    movel(p[x_c + -0.037960, y_c + 0.070717, z_c, rx, ry, rz], a, v)
    movel(p[x_c + -0.038280, y_c + 0.070511, z_c, rx, ry, rz], a, v)
    movel(p[x_c + -0.038598, y_c + 0.070300, z_c, rx, ry, rz], a, v)
    movel(p[x_c + -0.038913, y_c + 0.070083, z_c, rx, ry, rz], a, v)
    movel(p[x_c + -0.039226, y_c + 0.069859, z_c, rx, ry, rz], a, v)
    movel(p[x_c + -0.039535, y_c + 0.069631, z_c, rx, ry, rz], a, v)
    movel(p[x_c + -0.039842, y_c + 0.069396, z_c, rx, ry, rz], a, v)
    movel(p[x_c + -0.040146, y_c + 0.069155, z_c, rx, ry, rz], a, v)
    movel(p[x_c + -0.040448, y_c + 0.068909, z_c, rx, ry, rz], a, v)
    movel(p[x_c + -0.040746, y_c + 0.068657, z_c, rx, ry, rz], a, v)
    movel(p[x_c + -0.041042, y_c + 0.068400, z_c, rx, ry, rz], a, v)
    movel(p[x_c + -0.041335, y_c + 0.068137, z_c, rx, ry, rz], a, v)
    movel(p[x_c + -0.041625, y_c + 0.067868, z_c, rx, ry, rz], a, v)
    movel(p[x_c + -0.041912, y_c + 0.067594, z_c, rx, ry, rz], a, v)
    movel(p[x_c + -0.042196, y_c + 0.067314, z_c, rx, ry, rz], a, v)
    movel(p[x_c + -0.042477, y_c + 0.067029, z_c, rx, ry, rz], a, v)
    movel(p[x_c + -0.042756, y_c + 0.066738, z_c, rx, ry, rz], a, v)
    movel(p[x_c + -0.043031, y_c + 0.066441, z_c, rx, ry, rz], a, v)
    movel(p[x_c + -0.043303, y_c + 0.066140, z_c, rx, ry, rz], a, v)
    movel(p[x_c + -0.043572, y_c + 0.065832, z_c, rx, ry, rz], a, v)
    movel(p[x_c + -0.043838, y_c + 0.065520, z_c, rx, ry, rz], a, v)
    movel(p[x_c + -0.044100, y_c + 0.065202, z_c, rx, ry, rz], a, v)
    movel(p[x_c + -0.044360, y_c + 0.064879, z_c, rx, ry, rz], a, v)
    movel(p[x_c + -0.044616, y_c + 0.064550, z_c, rx, ry, rz], a, v)
    movel(p[x_c + -0.044870, y_c + 0.064217, z_c, rx, ry, rz], a, v)
    movel(p[x_c + -0.045120, y_c + 0.063877, z_c, rx, ry, rz], a, v)
    movel(p[x_c + -0.045366, y_c + 0.063533, z_c, rx, ry, rz], a, v)
    movel(p[x_c + -0.045610, y_c + 0.063184, z_c, rx, ry, rz], a, v)
    movel(p[x_c + -0.045850, y_c + 0.062829, z_c, rx, ry, rz], a, v)
    movel(p[x_c + -0.046087, y_c + 0.062470, z_c, rx, ry, rz], a, v)
    movel(p[x_c + -0.046320, y_c + 0.062105, z_c, rx, ry, rz], a, v)
    movel(p[x_c + -0.046550, y_c + 0.061735, z_c, rx, ry, rz], a, v)
    movel(p[x_c + -0.046776, y_c + 0.061360, z_c, rx, ry, rz], a, v)
    movel(p[x_c + -0.046999, y_c + 0.060980, z_c, rx, ry, rz], a, v)
    movel(p[x_c + -0.047219, y_c + 0.060595, z_c, rx, ry, rz], a, v)
    movel(p[x_c + -0.047435, y_c + 0.060205, z_c, rx, ry, rz], a, v)
    movel(p[x_c + -0.047648, y_c + 0.059810, z_c, rx, ry, rz], a, v)
    movel(p[x_c + -0.047857, y_c + 0.059410, z_c, rx, ry, rz], a, v)
    movel(p[x_c + -0.048062, y_c + 0.059006, z_c, rx, ry, rz], a, v)
    movel(p[x_c + -0.048264, y_c + 0.058596, z_c, rx, ry, rz], a, v)
    movel(p[x_c + -0.048462, y_c + 0.058182, z_c, rx, ry, rz], a, v)
    movel(p[x_c + -0.048462, y_c + 0.058182, z_c, rx, ry, rz], a, v)
    movel(p[x_c + -0.048836, y_c + 0.057374, z_c, rx, ry, rz], a, v)
    movel(p[x_c + -0.049201, y_c + 0.056551, z_c, rx, ry, rz], a, v)
    movel(p[x_c + -0.049559, y_c + 0.055714, z_c, rx, ry, rz], a, v)
    movel(p[x_c + -0.049909, y_c + 0.054862, z_c, rx, ry, rz], a, v)
    movel(p[x_c + -0.050251, y_c + 0.053997, z_c, rx, ry, rz], a, v)
    movel(p[x_c + -0.050586, y_c + 0.053117, z_c, rx, ry, rz], a, v)
    movel(p[x_c + -0.050912, y_c + 0.052224, z_c, rx, ry, rz], a, v)
    movel(p[x_c + -0.051231, y_c + 0.051318, z_c, rx, ry, rz], a, v)
    movel(p[x_c + -0.051541, y_c + 0.050399, z_c, rx, ry, rz], a, v)
    movel(p[x_c + -0.051843, y_c + 0.049467, z_c, rx, ry, rz], a, v)
    movel(p[x_c + -0.052138, y_c + 0.048523, z_c, rx, ry, rz], a, v)
    movel(p[x_c + -0.052424, y_c + 0.047567, z_c, rx, ry, rz], a, v)
    movel(p[x_c + -0.052702, y_c + 0.046599, z_c, rx, ry, rz], a, v)
    movel(p[x_c + -0.052971, y_c + 0.045619, z_c, rx, ry, rz], a, v)
    movel(p[x_c + -0.053233, y_c + 0.044627, z_c, rx, ry, rz], a, v)
    movel(p[x_c + -0.053486, y_c + 0.043625, z_c, rx, ry, rz], a, v)
    movel(p[x_c + -0.053730, y_c + 0.042612, z_c, rx, ry, rz], a, v)
    movel(p[x_c + -0.053967, y_c + 0.041588, z_c, rx, ry, rz], a, v)
    movel(p[x_c + -0.054195, y_c + 0.040554, z_c, rx, ry, rz], a, v)
    movel(p[x_c + -0.054414, y_c + 0.039510, z_c, rx, ry, rz], a, v)
    movel(p[x_c + -0.054625, y_c + 0.038456, z_c, rx, ry, rz], a, v)
    movel(p[x_c + -0.054827, y_c + 0.037393, z_c, rx, ry, rz], a, v)
    movel(p[x_c + -0.055021, y_c + 0.036320, z_c, rx, ry, rz], a, v)
    movel(p[x_c + -0.055206, y_c + 0.035238, z_c, rx, ry, rz], a, v)
    movel(p[x_c + -0.055382, y_c + 0.034148, z_c, rx, ry, rz], a, v)
    movel(p[x_c + -0.055550, y_c + 0.033049, z_c, rx, ry, rz], a, v)
    movel(p[x_c + -0.055709, y_c + 0.031942, z_c, rx, ry, rz], a, v)
    movel(p[x_c + -0.055859, y_c + 0.030827, z_c, rx, ry, rz], a, v)
    movel(p[x_c + -0.056000, y_c + 0.029705, z_c, rx, ry, rz], a, v)
    movel(p[x_c + -0.056132, y_c + 0.028575, z_c, rx, ry, rz], a, v)
    movel(p[x_c + -0.056255, y_c + 0.027438, z_c, rx, ry, rz], a, v)
    movel(p[x_c + -0.056369, y_c + 0.026294, z_c, rx, ry, rz], a, v)
    movel(p[x_c + -0.056475, y_c + 0.025143, z_c, rx, ry, rz], a, v)
    movel(p[x_c + -0.056571, y_c + 0.023986, z_c, rx, ry, rz], a, v)
    movel(p[x_c + -0.056658, y_c + 0.022823, z_c, rx, ry, rz], a, v)
    movel(p[x_c + -0.056735, y_c + 0.021654, z_c, rx, ry, rz], a, v)
    movel(p[x_c + -0.056804, y_c + 0.020480, z_c, rx, ry, rz], a, v)
    movel(p[x_c + -0.056863, y_c + 0.019301, z_c, rx, ry, rz], a, v)
    movel(p[x_c + -0.056913, y_c + 0.018116, z_c, rx, ry, rz], a, v)
    movel(p[x_c + -0.056954, y_c + 0.016927, z_c, rx, ry, rz], a, v)
    movel(p[x_c + -0.056985, y_c + 0.015733, z_c, rx, ry, rz], a, v)
    movel(p[x_c + -0.057007, y_c + 0.014535, z_c, rx, ry, rz], a, v)
    movel(p[x_c + -0.057019, y_c + 0.013333, z_c, rx, ry, rz], a, v)
    movel(p[x_c + -0.057022, y_c + 0.012127, z_c, rx, ry, rz], a, v)
    movel(p[x_c + -0.057015, y_c + 0.010918, z_c, rx, ry, rz], a, v)
    movel(p[x_c + -0.056999, y_c + 0.009706, z_c, rx, ry, rz], a, v)
    movel(p[x_c + -0.056973, y_c + 0.008491, z_c, rx, ry, rz], a, v)
    movel(p[x_c + -0.056938, y_c + 0.007273, z_c, rx, ry, rz], a, v)
    movel(p[x_c + -0.056892, y_c + 0.006053, z_c, rx, ry, rz], a, v)
    movel(p[x_c + -0.056892, y_c + 0.006053, z_c, rx, ry, rz], a, v)
    movel(p[x_c + -0.056865, y_c + 0.005424, z_c, rx, ry, rz], a, v)
    movel(p[x_c + -0.056837, y_c + 0.004798, z_c, rx, ry, rz], a, v)
    movel(p[x_c + -0.056806, y_c + 0.004175, z_c, rx, ry, rz], a, v)
    movel(p[x_c + -0.056774, y_c + 0.003554, z_c, rx, ry, rz], a, v)
    movel(p[x_c + -0.056740, y_c + 0.002935, z_c, rx, ry, rz], a, v)
    movel(p[x_c + -0.056704, y_c + 0.002319, z_c, rx, ry, rz], a, v)
    movel(p[x_c + -0.056666, y_c + 0.001705, z_c, rx, ry, rz], a, v)
    movel(p[x_c + -0.056627, y_c + 0.001093, z_c, rx, ry, rz], a, v)
    movel(p[x_c + -0.056585, y_c + 0.000483, z_c, rx, ry, rz], a, v)
    movel(p[x_c + -0.056542, y_c + -0.000124, z_c, rx, ry, rz], a, v)
    movel(p[x_c + -0.056497, y_c + -0.000730, z_c, rx, ry, rz], a, v)
    movel(p[x_c + -0.056450, y_c + -0.001334, z_c, rx, ry, rz], a, v)
    movel(p[x_c + -0.056401, y_c + -0.001936, z_c, rx, ry, rz], a, v)
    movel(p[x_c + -0.056350, y_c + -0.002536, z_c, rx, ry, rz], a, v)
    movel(p[x_c + -0.056297, y_c + -0.003135, z_c, rx, ry, rz], a, v)
    movel(p[x_c + -0.056242, y_c + -0.003732, z_c, rx, ry, rz], a, v)
    movel(p[x_c + -0.056185, y_c + -0.004328, z_c, rx, ry, rz], a, v)
    movel(p[x_c + -0.056127, y_c + -0.004922, z_c, rx, ry, rz], a, v)
    movel(p[x_c + -0.056066, y_c + -0.005515, z_c, rx, ry, rz], a, v)
    movel(p[x_c + -0.056003, y_c + -0.006106, z_c, rx, ry, rz], a, v)
    movel(p[x_c + -0.055939, y_c + -0.006697, z_c, rx, ry, rz], a, v)
    movel(p[x_c + -0.055872, y_c + -0.007286, z_c, rx, ry, rz], a, v)
    movel(p[x_c + -0.055803, y_c + -0.007874, z_c, rx, ry, rz], a, v)
    movel(p[x_c + -0.055733, y_c + -0.008462, z_c, rx, ry, rz], a, v)
    movel(p[x_c + -0.055660, y_c + -0.009048, z_c, rx, ry, rz], a, v)
    movel(p[x_c + -0.055586, y_c + -0.009634, z_c, rx, ry, rz], a, v)
    movel(p[x_c + -0.055509, y_c + -0.010219, z_c, rx, ry, rz], a, v)
    movel(p[x_c + -0.055430, y_c + -0.010803, z_c, rx, ry, rz], a, v)
    movel(p[x_c + -0.055350, y_c + -0.011387, z_c, rx, ry, rz], a, v)
    movel(p[x_c + -0.055267, y_c + -0.011970, z_c, rx, ry, rz], a, v)
    movel(p[x_c + -0.055182, y_c + -0.012553, z_c, rx, ry, rz], a, v)
    movel(p[x_c + -0.055095, y_c + -0.013135, z_c, rx, ry, rz], a, v)
    movel(p[x_c + -0.055006, y_c + -0.013717, z_c, rx, ry, rz], a, v)
    movel(p[x_c + -0.054915, y_c + -0.014299, z_c, rx, ry, rz], a, v)
    movel(p[x_c + -0.054821, y_c + -0.014881, z_c, rx, ry, rz], a, v)
    movel(p[x_c + -0.054726, y_c + -0.015463, z_c, rx, ry, rz], a, v)
    movel(p[x_c + -0.054628, y_c + -0.016045, z_c, rx, ry, rz], a, v)
    movel(p[x_c + -0.054529, y_c + -0.016627, z_c, rx, ry, rz], a, v)
    movel(p[x_c + -0.054427, y_c + -0.017209, z_c, rx, ry, rz], a, v)
    movel(p[x_c + -0.054323, y_c + -0.017791, z_c, rx, ry, rz], a, v)
    movel(p[x_c + -0.054217, y_c + -0.018374, z_c, rx, ry, rz], a, v)
    movel(p[x_c + -0.054108, y_c + -0.018957, z_c, rx, ry, rz], a, v)
    movel(p[x_c + -0.053998, y_c + -0.019541, z_c, rx, ry, rz], a, v)
    movel(p[x_c + -0.053885, y_c + -0.020125, z_c, rx, ry, rz], a, v)
    movel(p[x_c + -0.053770, y_c + -0.020710, z_c, rx, ry, rz], a, v)
    movel(p[x_c + -0.053653, y_c + -0.021296, z_c, rx, ry, rz], a, v)
    movel(p[x_c + -0.053534, y_c + -0.021882, z_c, rx, ry, rz], a, v)
    movel(p[x_c + -0.053412, y_c + -0.022470, z_c, rx, ry, rz], a, v)
    movel(p[x_c + -0.053288, y_c + -0.023058, z_c, rx, ry, rz], a, v)
    movel(p[x_c + -0.053288, y_c + -0.023058, z_c, rx, ry, rz], a, v)
    movel(p[x_c + -0.053049, y_c + -0.024173, z_c, rx, ry, rz], a, v)
    movel(p[x_c + -0.052804, y_c + -0.025284, z_c, rx, ry, rz], a, v)
    movel(p[x_c + -0.052555, y_c + -0.026393, z_c, rx, ry, rz], a, v)
    movel(p[x_c + -0.052300, y_c + -0.027499, z_c, rx, ry, rz], a, v)
    movel(p[x_c + -0.052040, y_c + -0.028602, z_c, rx, ry, rz], a, v)
    movel(p[x_c + -0.051775, y_c + -0.029701, z_c, rx, ry, rz], a, v)
    movel(p[x_c + -0.051505, y_c + -0.030798, z_c, rx, ry, rz], a, v)
    movel(p[x_c + -0.051230, y_c + -0.031891, z_c, rx, ry, rz], a, v)
    movel(p[x_c + -0.050950, y_c + -0.032980, z_c, rx, ry, rz], a, v)
    movel(p[x_c + -0.050666, y_c + -0.034067, z_c, rx, ry, rz], a, v)
    movel(p[x_c + -0.050376, y_c + -0.035150, z_c, rx, ry, rz], a, v)
    movel(p[x_c + -0.050081, y_c + -0.036229, z_c, rx, ry, rz], a, v)
    movel(p[x_c + -0.049781, y_c + -0.037305, z_c, rx, ry, rz], a, v)
    movel(p[x_c + -0.049477, y_c + -0.038377, z_c, rx, ry, rz], a, v)
    movel(p[x_c + -0.049168, y_c + -0.039446, z_c, rx, ry, rz], a, v)
    movel(p[x_c + -0.048853, y_c + -0.040510, z_c, rx, ry, rz], a, v)
    movel(p[x_c + -0.048534, y_c + -0.041571, z_c, rx, ry, rz], a, v)
    movel(p[x_c + -0.048210, y_c + -0.042629, z_c, rx, ry, rz], a, v)
    movel(p[x_c + -0.047882, y_c + -0.043682, z_c, rx, ry, rz], a, v)
    movel(p[x_c + -0.047548, y_c + -0.044731, z_c, rx, ry, rz], a, v)
    movel(p[x_c + -0.047210, y_c + -0.045777, z_c, rx, ry, rz], a, v)
    movel(p[x_c + -0.046867, y_c + -0.046818, z_c, rx, ry, rz], a, v)
    movel(p[x_c + -0.046520, y_c + -0.047855, z_c, rx, ry, rz], a, v)
    movel(p[x_c + -0.046167, y_c + -0.048888, z_c, rx, ry, rz], a, v)
    movel(p[x_c + -0.045811, y_c + -0.049917, z_c, rx, ry, rz], a, v)
    movel(p[x_c + -0.045449, y_c + -0.050941, z_c, rx, ry, rz], a, v)
    movel(p[x_c + -0.045083, y_c + -0.051961, z_c, rx, ry, rz], a, v)
    movel(p[x_c + -0.044712, y_c + -0.052977, z_c, rx, ry, rz], a, v)
    movel(p[x_c + -0.044336, y_c + -0.053988, z_c, rx, ry, rz], a, v)
    movel(p[x_c + -0.043956, y_c + -0.054994, z_c, rx, ry, rz], a, v)
    movel(p[x_c + -0.043572, y_c + -0.055997, z_c, rx, ry, rz], a, v)
    movel(p[x_c + -0.043183, y_c + -0.056994, z_c, rx, ry, rz], a, v)
    movel(p[x_c + -0.042789, y_c + -0.057987, z_c, rx, ry, rz], a, v)
    movel(p[x_c + -0.042391, y_c + -0.058975, z_c, rx, ry, rz], a, v)
    movel(p[x_c + -0.041989, y_c + -0.059958, z_c, rx, ry, rz], a, v)
    movel(p[x_c + -0.041582, y_c + -0.060936, z_c, rx, ry, rz], a, v)
    movel(p[x_c + -0.041170, y_c + -0.061910, z_c, rx, ry, rz], a, v)
    movel(p[x_c + -0.040754, y_c + -0.062878, z_c, rx, ry, rz], a, v)
    movel(p[x_c + -0.040334, y_c + -0.063842, z_c, rx, ry, rz], a, v)
    movel(p[x_c + -0.039909, y_c + -0.064800, z_c, rx, ry, rz], a, v)
    movel(p[x_c + -0.039480, y_c + -0.065753, z_c, rx, ry, rz], a, v)
    movel(p[x_c + -0.039047, y_c + -0.066701, z_c, rx, ry, rz], a, v)
    movel(p[x_c + -0.038610, y_c + -0.067644, z_c, rx, ry, rz], a, v)
    movel(p[x_c + -0.038168, y_c + -0.068581, z_c, rx, ry, rz], a, v)
    movel(p[x_c + -0.037721, y_c + -0.069513, z_c, rx, ry, rz], a, v)
    movel(p[x_c + -0.037271, y_c + -0.070440, z_c, rx, ry, rz], a, v)
    movel(p[x_c + -0.036816, y_c + -0.071361, z_c, rx, ry, rz], a, v)
    movel(p[x_c + -0.036357, y_c + -0.072277, z_c, rx, ry, rz], a, v)
    movel(p[x_c + -0.035894, y_c + -0.073187, z_c, rx, ry, rz], a, v)
    movel(p[x_c + -0.035894, y_c + -0.073187, z_c, rx, ry, rz], a, v)
    movel(p[x_c + -0.035415, y_c + -0.074118, z_c, rx, ry, rz], a, v)
    movel(p[x_c + -0.034944, y_c + -0.075025, z_c, rx, ry, rz], a, v)
    movel(p[x_c + -0.034481, y_c + -0.075907, z_c, rx, ry, rz], a, v)
    movel(p[x_c + -0.034027, y_c + -0.076765, z_c, rx, ry, rz], a, v)
    movel(p[x_c + -0.033579, y_c + -0.077599, z_c, rx, ry, rz], a, v)
    movel(p[x_c + -0.033140, y_c + -0.078411, z_c, rx, ry, rz], a, v)
    movel(p[x_c + -0.032707, y_c + -0.079199, z_c, rx, ry, rz], a, v)
    movel(p[x_c + -0.032280, y_c + -0.079966, z_c, rx, ry, rz], a, v)
    movel(p[x_c + -0.031860, y_c + -0.080711, z_c, rx, ry, rz], a, v)
    movel(p[x_c + -0.031445, y_c + -0.081434, z_c, rx, ry, rz], a, v)
    movel(p[x_c + -0.031036, y_c + -0.082137, z_c, rx, ry, rz], a, v)
    movel(p[x_c + -0.030632, y_c + -0.082819, z_c, rx, ry, rz], a, v)
    movel(p[x_c + -0.030233, y_c + -0.083481, z_c, rx, ry, rz], a, v)
    movel(p[x_c + -0.029838, y_c + -0.084124, z_c, rx, ry, rz], a, v)
    movel(p[x_c + -0.029447, y_c + -0.084747, z_c, rx, ry, rz], a, v)
    movel(p[x_c + -0.029059, y_c + -0.085352, z_c, rx, ry, rz], a, v)
    movel(p[x_c + -0.028675, y_c + -0.085939, z_c, rx, ry, rz], a, v)
    movel(p[x_c + -0.028293, y_c + -0.086508, z_c, rx, ry, rz], a, v)
    movel(p[x_c + -0.027914, y_c + -0.087059, z_c, rx, ry, rz], a, v)
    movel(p[x_c + -0.027537, y_c + -0.087594, z_c, rx, ry, rz], a, v)
    movel(p[x_c + -0.027162, y_c + -0.088113, z_c, rx, ry, rz], a, v)
    movel(p[x_c + -0.026789, y_c + -0.088615, z_c, rx, ry, rz], a, v)
    movel(p[x_c + -0.026416, y_c + -0.089102, z_c, rx, ry, rz], a, v)
    movel(p[x_c + -0.026044, y_c + -0.089574, z_c, rx, ry, rz], a, v)
    movel(p[x_c + -0.025673, y_c + -0.090032, z_c, rx, ry, rz], a, v)
    movel(p[x_c + -0.025301, y_c + -0.090475, z_c, rx, ry, rz], a, v)
    movel(p[x_c + -0.024929, y_c + -0.090905, z_c, rx, ry, rz], a, v)
    movel(p[x_c + -0.024556, y_c + -0.091321, z_c, rx, ry, rz], a, v)
    movel(p[x_c + -0.024182, y_c + -0.091724, z_c, rx, ry, rz], a, v)
    movel(p[x_c + -0.023806, y_c + -0.092115, z_c, rx, ry, rz], a, v)
    movel(p[x_c + -0.023429, y_c + -0.092495, z_c, rx, ry, rz], a, v)
    movel(p[x_c + -0.023050, y_c + -0.092862, z_c, rx, ry, rz], a, v)
    movel(p[x_c + -0.022667, y_c + -0.093219, z_c, rx, ry, rz], a, v)
    movel(p[x_c + -0.022282, y_c + -0.093565, z_c, rx, ry, rz], a, v)
    movel(p[x_c + -0.021894, y_c + -0.093901, z_c, rx, ry, rz], a, v)
    movel(p[x_c + -0.021502, y_c + -0.094228, z_c, rx, ry, rz], a, v)
    movel(p[x_c + -0.021105, y_c + -0.094545, z_c, rx, ry, rz], a, v)
    movel(p[x_c + -0.020705, y_c + -0.094853, z_c, rx, ry, rz], a, v)
    movel(p[x_c + -0.020299, y_c + -0.095153, z_c, rx, ry, rz], a, v)
    movel(p[x_c + -0.019889, y_c + -0.095446, z_c, rx, ry, rz], a, v)
    movel(p[x_c + -0.019473, y_c + -0.095730, z_c, rx, ry, rz], a, v)
    movel(p[x_c + -0.019051, y_c + -0.096008, z_c, rx, ry, rz], a, v)
    movel(p[x_c + -0.018622, y_c + -0.096279, z_c, rx, ry, rz], a, v)
    movel(p[x_c + -0.018188, y_c + -0.096544, z_c, rx, ry, rz], a, v)
    movel(p[x_c + -0.017746, y_c + -0.096804, z_c, rx, ry, rz], a, v)
    movel(p[x_c + -0.017297, y_c + -0.097058, z_c, rx, ry, rz], a, v)
    movel(p[x_c + -0.016840, y_c + -0.097308, z_c, rx, ry, rz], a, v)
    movel(p[x_c + -0.016375, y_c + -0.097553, z_c, rx, ry, rz], a, v)
    movel(p[x_c + -0.015902, y_c + -0.097795, z_c, rx, ry, rz], a, v)
    movel(p[x_c + -0.015902, y_c + -0.097795, z_c, rx, ry, rz], a, v)
    movel(p[x_c + -0.015678, y_c + -0.097906, z_c, rx, ry, rz], a, v)
    movel(p[x_c + -0.015447, y_c + -0.098017, z_c, rx, ry, rz], a, v)
    movel(p[x_c + -0.015209, y_c + -0.098129, z_c, rx, ry, rz], a, v)
    movel(p[x_c + -0.014967, y_c + -0.098241, z_c, rx, ry, rz], a, v)
    movel(p[x_c + -0.014718, y_c + -0.098354, z_c, rx, ry, rz], a, v)
    movel(p[x_c + -0.014465, y_c + -0.098466, z_c, rx, ry, rz], a, v)
    movel(p[x_c + -0.014207, y_c + -0.098578, z_c, rx, ry, rz], a, v)
    movel(p[x_c + -0.013944, y_c + -0.098690, z_c, rx, ry, rz], a, v)
    movel(p[x_c + -0.013678, y_c + -0.098801, z_c, rx, ry, rz], a, v)
    movel(p[x_c + -0.013408, y_c + -0.098912, z_c, rx, ry, rz], a, v)
    movel(p[x_c + -0.013135, y_c + -0.099023, z_c, rx, ry, rz], a, v)
    movel(p[x_c + -0.012859, y_c + -0.099132, z_c, rx, ry, rz], a, v)
    movel(p[x_c + -0.012580, y_c + -0.099241, z_c, rx, ry, rz], a, v)
    movel(p[x_c + -0.012299, y_c + -0.099349, z_c, rx, ry, rz], a, v)
    movel(p[x_c + -0.012016, y_c + -0.099456, z_c, rx, ry, rz], a, v)
    movel(p[x_c + -0.011732, y_c + -0.099561, z_c, rx, ry, rz], a, v)
    movel(p[x_c + -0.011447, y_c + -0.099666, z_c, rx, ry, rz], a, v)
    movel(p[x_c + -0.011161, y_c + -0.099768, z_c, rx, ry, rz], a, v)
    movel(p[x_c + -0.010874, y_c + -0.099870, z_c, rx, ry, rz], a, v)
    movel(p[x_c + -0.010588, y_c + -0.099970, z_c, rx, ry, rz], a, v)
    movel(p[x_c + -0.010302, y_c + -0.100068, z_c, rx, ry, rz], a, v)
    movel(p[x_c + -0.010016, y_c + -0.100164, z_c, rx, ry, rz], a, v)
    movel(p[x_c + -0.009732, y_c + -0.100258, z_c, rx, ry, rz], a, v)
    movel(p[x_c + -0.009449, y_c + -0.100350, z_c, rx, ry, rz], a, v)
    movel(p[x_c + -0.009168, y_c + -0.100440, z_c, rx, ry, rz], a, v)
    movel(p[x_c + -0.008888, y_c + -0.100527, z_c, rx, ry, rz], a, v)
    movel(p[x_c + -0.008612, y_c + -0.100612, z_c, rx, ry, rz], a, v)
    movel(p[x_c + -0.008338, y_c + -0.100695, z_c, rx, ry, rz], a, v)
    movel(p[x_c + -0.008067, y_c + -0.100775, z_c, rx, ry, rz], a, v)
    movel(p[x_c + -0.007800, y_c + -0.100852, z_c, rx, ry, rz], a, v)
    movel(p[x_c + -0.007537, y_c + -0.100926, z_c, rx, ry, rz], a, v)
    movel(p[x_c + -0.007278, y_c + -0.100997, z_c, rx, ry, rz], a, v)
    movel(p[x_c + -0.007024, y_c + -0.101065, z_c, rx, ry, rz], a, v)
    movel(p[x_c + -0.006775, y_c + -0.101130, z_c, rx, ry, rz], a, v)
    movel(p[x_c + -0.006531, y_c + -0.101192, z_c, rx, ry, rz], a, v)
    movel(p[x_c + -0.006293, y_c + -0.101250, z_c, rx, ry, rz], a, v)
    movel(p[x_c + -0.006060, y_c + -0.101304, z_c, rx, ry, rz], a, v)
    movel(p[x_c + -0.005835, y_c + -0.101355, z_c, rx, ry, rz], a, v)
    movel(p[x_c + -0.005616, y_c + -0.101402, z_c, rx, ry, rz], a, v)
    movel(p[x_c + -0.005404, y_c + -0.101445, z_c, rx, ry, rz], a, v)
    movel(p[x_c + -0.005200, y_c + -0.101484, z_c, rx, ry, rz], a, v)
    movel(p[x_c + -0.005003, y_c + -0.101518, z_c, rx, ry, rz], a, v)
    movel(p[x_c + -0.004815, y_c + -0.101549, z_c, rx, ry, rz], a, v)
    movel(p[x_c + -0.004635, y_c + -0.101575, z_c, rx, ry, rz], a, v)
    movel(p[x_c + -0.004465, y_c + -0.101596, z_c, rx, ry, rz], a, v)
    movel(p[x_c + -0.004303, y_c + -0.101613, z_c, rx, ry, rz], a, v)
    movel(p[x_c + -0.004152, y_c + -0.101626, z_c, rx, ry, rz], a, v)
    movel(p[x_c + -0.004010, y_c + -0.101633, z_c, rx, ry, rz], a, v)
    movel(p[x_c + -0.003878, y_c + -0.101636, z_c, rx, ry, rz], a, v)
    movel(p[x_c + -0.003878, y_c + -0.101636, z_c, rx, ry, rz], a, v)
    movel(p[x_c + -0.003761, y_c + -0.101634, z_c, rx, ry, rz], a, v)
    movel(p[x_c + -0.003645, y_c + -0.101629, z_c, rx, ry, rz], a, v)
    movel(p[x_c + -0.003531, y_c + -0.101621, z_c, rx, ry, rz], a, v)
    movel(p[x_c + -0.003417, y_c + -0.101609, z_c, rx, ry, rz], a, v)
    movel(p[x_c + -0.003305, y_c + -0.101595, z_c, rx, ry, rz], a, v)
    movel(p[x_c + -0.003195, y_c + -0.101577, z_c, rx, ry, rz], a, v)
    movel(p[x_c + -0.003086, y_c + -0.101556, z_c, rx, ry, rz], a, v)
    movel(p[x_c + -0.002978, y_c + -0.101532, z_c, rx, ry, rz], a, v)
    movel(p[x_c + -0.002872, y_c + -0.101505, z_c, rx, ry, rz], a, v)
    movel(p[x_c + -0.002767, y_c + -0.101474, z_c, rx, ry, rz], a, v)
    movel(p[x_c + -0.002664, y_c + -0.101441, z_c, rx, ry, rz], a, v)
    movel(p[x_c + -0.002563, y_c + -0.101405, z_c, rx, ry, rz], a, v)
    movel(p[x_c + -0.002463, y_c + -0.101366, z_c, rx, ry, rz], a, v)
    movel(p[x_c + -0.002365, y_c + -0.101324, z_c, rx, ry, rz], a, v)
    movel(p[x_c + -0.002269, y_c + -0.101279, z_c, rx, ry, rz], a, v)
    movel(p[x_c + -0.002174, y_c + -0.101231, z_c, rx, ry, rz], a, v)
    movel(p[x_c + -0.002081, y_c + -0.101181, z_c, rx, ry, rz], a, v)
    movel(p[x_c + -0.001990, y_c + -0.101127, z_c, rx, ry, rz], a, v)
    movel(p[x_c + -0.001901, y_c + -0.101071, z_c, rx, ry, rz], a, v)
    movel(p[x_c + -0.001813, y_c + -0.101012, z_c, rx, ry, rz], a, v)
    movel(p[x_c + -0.001728, y_c + -0.100951, z_c, rx, ry, rz], a, v)
    movel(p[x_c + -0.001645, y_c + -0.100887, z_c, rx, ry, rz], a, v)
    movel(p[x_c + -0.001563, y_c + -0.100820, z_c, rx, ry, rz], a, v)
    movel(p[x_c + -0.001484, y_c + -0.100750, z_c, rx, ry, rz], a, v)
    movel(p[x_c + -0.001406, y_c + -0.100678, z_c, rx, ry, rz], a, v)
    movel(p[x_c + -0.001331, y_c + -0.100604, z_c, rx, ry, rz], a, v)
    movel(p[x_c + -0.001258, y_c + -0.100527, z_c, rx, ry, rz], a, v)
    movel(p[x_c + -0.001187, y_c + -0.100447, z_c, rx, ry, rz], a, v)
    movel(p[x_c + -0.001118, y_c + -0.100365, z_c, rx, ry, rz], a, v)
    movel(p[x_c + -0.001051, y_c + -0.100281, z_c, rx, ry, rz], a, v)
    movel(p[x_c + -0.000987, y_c + -0.100194, z_c, rx, ry, rz], a, v)
    movel(p[x_c + -0.000924, y_c + -0.100105, z_c, rx, ry, rz], a, v)
    movel(p[x_c + -0.000865, y_c + -0.100014, z_c, rx, ry, rz], a, v)
    movel(p[x_c + -0.000807, y_c + -0.099920, z_c, rx, ry, rz], a, v)
    movel(p[x_c + -0.000752, y_c + -0.099824, z_c, rx, ry, rz], a, v)
    movel(p[x_c + -0.000699, y_c + -0.099726, z_c, rx, ry, rz], a, v)
    movel(p[x_c + -0.000649, y_c + -0.099626, z_c, rx, ry, rz], a, v)
    movel(p[x_c + -0.000602, y_c + -0.099524, z_c, rx, ry, rz], a, v)
    movel(p[x_c + -0.000556, y_c + -0.099419, z_c, rx, ry, rz], a, v)
    movel(p[x_c + -0.000514, y_c + -0.099312, z_c, rx, ry, rz], a, v)
    movel(p[x_c + -0.000474, y_c + -0.099204, z_c, rx, ry, rz], a, v)
    movel(p[x_c + -0.000436, y_c + -0.099093, z_c, rx, ry, rz], a, v)
    movel(p[x_c + -0.000402, y_c + -0.098980, z_c, rx, ry, rz], a, v)
    movel(p[x_c + -0.000370, y_c + -0.098865, z_c, rx, ry, rz], a, v)
    movel(p[x_c + -0.000340, y_c + -0.098749, z_c, rx, ry, rz], a, v)
    movel(p[x_c + -0.000314, y_c + -0.098630, z_c, rx, ry, rz], a, v)
    movel(p[x_c + -0.000290, y_c + -0.098510, z_c, rx, ry, rz], a, v)
    movel(p[x_c + -0.000269, y_c + -0.098387, z_c, rx, ry, rz], a, v)
    movel(p[x_c + -0.000251, y_c + -0.098263, z_c, rx, ry, rz], a, v)
    movel(p[x_c + -0.000251, y_c + -0.098263, z_c, rx, ry, rz], a, v)
    movel(p[x_c + -0.000107, y_c + -0.097177, z_c, rx, ry, rz], a, v)
    movel(p[x_c + -0.000107, y_c + -0.097177, z_c, rx, ry, rz], a, v)
    movel(p[x_c + 0.001456, y_c + -0.097998, z_c, rx, ry, rz], a, v)
    movel(p[x_c + 0.001456, y_c + -0.097998, z_c, rx, ry, rz], a, v)
    movel(p[x_c + 0.001663, y_c + -0.098109, z_c, rx, ry, rz], a, v)
    movel(p[x_c + 0.001866, y_c + -0.098221, z_c, rx, ry, rz], a, v)
    movel(p[x_c + 0.002064, y_c + -0.098333, z_c, rx, ry, rz], a, v)
    movel(p[x_c + 0.002258, y_c + -0.098447, z_c, rx, ry, rz], a, v)
    movel(p[x_c + 0.002446, y_c + -0.098562, z_c, rx, ry, rz], a, v)
    movel(p[x_c + 0.002631, y_c + -0.098678, z_c, rx, ry, rz], a, v)
    movel(p[x_c + 0.002811, y_c + -0.098795, z_c, rx, ry, rz], a, v)
    movel(p[x_c + 0.002987, y_c + -0.098914, z_c, rx, ry, rz], a, v)
    movel(p[x_c + 0.003158, y_c + -0.099035, z_c, rx, ry, rz], a, v)
    movel(p[x_c + 0.003325, y_c + -0.099157, z_c, rx, ry, rz], a, v)
    movel(p[x_c + 0.003488, y_c + -0.099280, z_c, rx, ry, rz], a, v)
    movel(p[x_c + 0.003647, y_c + -0.099406, z_c, rx, ry, rz], a, v)
    movel(p[x_c + 0.003802, y_c + -0.099533, z_c, rx, ry, rz], a, v)
    movel(p[x_c + 0.003953, y_c + -0.099663, z_c, rx, ry, rz], a, v)
    movel(p[x_c + 0.004100, y_c + -0.099794, z_c, rx, ry, rz], a, v)
    movel(p[x_c + 0.004243, y_c + -0.099928, z_c, rx, ry, rz], a, v)
    movel(p[x_c + 0.004383, y_c + -0.100064, z_c, rx, ry, rz], a, v)
    movel(p[x_c + 0.004518, y_c + -0.100202, z_c, rx, ry, rz], a, v)
    movel(p[x_c + 0.004650, y_c + -0.100342, z_c, rx, ry, rz], a, v)
    movel(p[x_c + 0.004779, y_c + -0.100485, z_c, rx, ry, rz], a, v)
    movel(p[x_c + 0.004904, y_c + -0.100631, z_c, rx, ry, rz], a, v)
    movel(p[x_c + 0.005025, y_c + -0.100779, z_c, rx, ry, rz], a, v)
    movel(p[x_c + 0.005143, y_c + -0.100930, z_c, rx, ry, rz], a, v)
    movel(p[x_c + 0.005258, y_c + -0.101084, z_c, rx, ry, rz], a, v)
    movel(p[x_c + 0.005369, y_c + -0.101240, z_c, rx, ry, rz], a, v)
    movel(p[x_c + 0.005477, y_c + -0.101400, z_c, rx, ry, rz], a, v)
    movel(p[x_c + 0.005582, y_c + -0.101563, z_c, rx, ry, rz], a, v)
    movel(p[x_c + 0.005684, y_c + -0.101729, z_c, rx, ry, rz], a, v)
    movel(p[x_c + 0.005782, y_c + -0.101898, z_c, rx, ry, rz], a, v)
    movel(p[x_c + 0.005878, y_c + -0.102071, z_c, rx, ry, rz], a, v)
    movel(p[x_c + 0.005971, y_c + -0.102247, z_c, rx, ry, rz], a, v)
    movel(p[x_c + 0.006061, y_c + -0.102426, z_c, rx, ry, rz], a, v)
    movel(p[x_c + 0.006148, y_c + -0.102609, z_c, rx, ry, rz], a, v)
    movel(p[x_c + 0.006232, y_c + -0.102796, z_c, rx, ry, rz], a, v)
    movel(p[x_c + 0.006314, y_c + -0.102987, z_c, rx, ry, rz], a, v)
    movel(p[x_c + 0.006393, y_c + -0.103181, z_c, rx, ry, rz], a, v)
    movel(p[x_c + 0.006470, y_c + -0.103380, z_c, rx, ry, rz], a, v)
    movel(p[x_c + 0.006544, y_c + -0.103582, z_c, rx, ry, rz], a, v)
    movel(p[x_c + 0.006615, y_c + -0.103789, z_c, rx, ry, rz], a, v)
    movel(p[x_c + 0.006685, y_c + -0.104000, z_c, rx, ry, rz], a, v)
    movel(p[x_c + 0.006751, y_c + -0.104215, z_c, rx, ry, rz], a, v)
    movel(p[x_c + 0.006816, y_c + -0.104434, z_c, rx, ry, rz], a, v)
    movel(p[x_c + 0.006879, y_c + -0.104658, z_c, rx, ry, rz], a, v)
    movel(p[x_c + 0.006939, y_c + -0.104887, z_c, rx, ry, rz], a, v)
    movel(p[x_c + 0.006997, y_c + -0.105120, z_c, rx, ry, rz], a, v)
    movel(p[x_c + 0.007054, y_c + -0.105358, z_c, rx, ry, rz], a, v)
    movel(p[x_c + 0.007108, y_c + -0.105601, z_c, rx, ry, rz], a, v)
    movel(p[x_c + 0.007160, y_c + -0.105848, z_c, rx, ry, rz], a, v)
    movel(p[x_c + 0.007211, y_c + -0.106101, z_c, rx, ry, rz], a, v)
    movel(p[x_c + 0.007211, y_c + -0.106101, z_c, rx, ry, rz], a, v)
    movel(p[x_c + 0.007250, y_c + -0.106301, z_c, rx, ry, rz], a, v)
    movel(p[x_c + 0.007288, y_c + -0.106493, z_c, rx, ry, rz], a, v)
    movel(p[x_c + 0.007324, y_c + -0.106677, z_c, rx, ry, rz], a, v)
    movel(p[x_c + 0.007359, y_c + -0.106853, z_c, rx, ry, rz], a, v)
    movel(p[x_c + 0.007393, y_c + -0.107022, z_c, rx, ry, rz], a, v)
    movel(p[x_c + 0.007426, y_c + -0.107184, z_c, rx, ry, rz], a, v)
    movel(p[x_c + 0.007457, y_c + -0.107338, z_c, rx, ry, rz], a, v)
    movel(p[x_c + 0.007488, y_c + -0.107485, z_c, rx, ry, rz], a, v)
    movel(p[x_c + 0.007518, y_c + -0.107626, z_c, rx, ry, rz], a, v)
    movel(p[x_c + 0.007547, y_c + -0.107760, z_c, rx, ry, rz], a, v)
    movel(p[x_c + 0.007576, y_c + -0.107887, z_c, rx, ry, rz], a, v)
    movel(p[x_c + 0.007604, y_c + -0.108008, z_c, rx, ry, rz], a, v)
    movel(p[x_c + 0.007631, y_c + -0.108122, z_c, rx, ry, rz], a, v)
    movel(p[x_c + 0.007658, y_c + -0.108230, z_c, rx, ry, rz], a, v)
    movel(p[x_c + 0.007685, y_c + -0.108333, z_c, rx, ry, rz], a, v)
    movel(p[x_c + 0.007711, y_c + -0.108429, z_c, rx, ry, rz], a, v)
    movel(p[x_c + 0.007737, y_c + -0.108520, z_c, rx, ry, rz], a, v)
    movel(p[x_c + 0.007763, y_c + -0.108606, z_c, rx, ry, rz], a, v)
    movel(p[x_c + 0.007790, y_c + -0.108686, z_c, rx, ry, rz], a, v)
    movel(p[x_c + 0.007816, y_c + -0.108760, z_c, rx, ry, rz], a, v)
    movel(p[x_c + 0.007842, y_c + -0.108830, z_c, rx, ry, rz], a, v)
    movel(p[x_c + 0.007868, y_c + -0.108895, z_c, rx, ry, rz], a, v)
    movel(p[x_c + 0.007895, y_c + -0.108955, z_c, rx, ry, rz], a, v)
    movel(p[x_c + 0.007922, y_c + -0.109010, z_c, rx, ry, rz], a, v)
    movel(p[x_c + 0.007950, y_c + -0.109061, z_c, rx, ry, rz], a, v)
    movel(p[x_c + 0.007978, y_c + -0.109108, z_c, rx, ry, rz], a, v)
    movel(p[x_c + 0.008007, y_c + -0.109151, z_c, rx, ry, rz], a, v)
    movel(p[x_c + 0.008037, y_c + -0.109189, z_c, rx, ry, rz], a, v)
    movel(p[x_c + 0.008067, y_c + -0.109224, z_c, rx, ry, rz], a, v)
    movel(p[x_c + 0.008099, y_c + -0.109255, z_c, rx, ry, rz], a, v)
    movel(p[x_c + 0.008131, y_c + -0.109282, z_c, rx, ry, rz], a, v)
    movel(p[x_c + 0.008164, y_c + -0.109306, z_c, rx, ry, rz], a, v)
    movel(p[x_c + 0.008198, y_c + -0.109327, z_c, rx, ry, rz], a, v)
    movel(p[x_c + 0.008234, y_c + -0.109345, z_c, rx, ry, rz], a, v)
    movel(p[x_c + 0.008271, y_c + -0.109359, z_c, rx, ry, rz], a, v)
    movel(p[x_c + 0.008309, y_c + -0.109371, z_c, rx, ry, rz], a, v)
    movel(p[x_c + 0.008349, y_c + -0.109380, z_c, rx, ry, rz], a, v)
    movel(p[x_c + 0.008390, y_c + -0.109387, z_c, rx, ry, rz], a, v)
    movel(p[x_c + 0.008433, y_c + -0.109392, z_c, rx, ry, rz], a, v)
    movel(p[x_c + 0.008478, y_c + -0.109394, z_c, rx, ry, rz], a, v)
    movel(p[x_c + 0.008524, y_c + -0.109394, z_c, rx, ry, rz], a, v)
    movel(p[x_c + 0.008573, y_c + -0.109393, z_c, rx, ry, rz], a, v)
    movel(p[x_c + 0.008623, y_c + -0.109389, z_c, rx, ry, rz], a, v)
    movel(p[x_c + 0.008675, y_c + -0.109384, z_c, rx, ry, rz], a, v)
    movel(p[x_c + 0.008730, y_c + -0.109378, z_c, rx, ry, rz], a, v)
    movel(p[x_c + 0.008786, y_c + -0.109370, z_c, rx, ry, rz], a, v)
    movel(p[x_c + 0.008845, y_c + -0.109361, z_c, rx, ry, rz], a, v)
    movel(p[x_c + 0.008907, y_c + -0.109352, z_c, rx, ry, rz], a, v)
    movel(p[x_c + 0.008970, y_c + -0.109341, z_c, rx, ry, rz], a, v)
    movel(p[x_c + 0.008970, y_c + -0.109341, z_c, rx, ry, rz], a, v)
    movel(p[x_c + 0.009063, y_c + -0.109327, z_c, rx, ry, rz], a, v)
    movel(p[x_c + 0.009156, y_c + -0.109315, z_c, rx, ry, rz], a, v)
    movel(p[x_c + 0.009248, y_c + -0.109306, z_c, rx, ry, rz], a, v)
    movel(p[x_c + 0.009340, y_c + -0.109299, z_c, rx, ry, rz], a, v)
    movel(p[x_c + 0.009431, y_c + -0.109295, z_c, rx, ry, rz], a, v)
    movel(p[x_c + 0.009523, y_c + -0.109294, z_c, rx, ry, rz], a, v)
    movel(p[x_c + 0.009614, y_c + -0.109296, z_c, rx, ry, rz], a, v)
    movel(p[x_c + 0.009705, y_c + -0.109301, z_c, rx, ry, rz], a, v)
    movel(p[x_c + 0.009797, y_c + -0.109308, z_c, rx, ry, rz], a, v)
    movel(p[x_c + 0.009888, y_c + -0.109318, z_c, rx, ry, rz], a, v)
    movel(p[x_c + 0.009979, y_c + -0.109331, z_c, rx, ry, rz], a, v)
    movel(p[x_c + 0.010071, y_c + -0.109347, z_c, rx, ry, rz], a, v)
    movel(p[x_c + 0.010163, y_c + -0.109366, z_c, rx, ry, rz], a, v)
    movel(p[x_c + 0.010255, y_c + -0.109388, z_c, rx, ry, rz], a, v)
    movel(p[x_c + 0.010347, y_c + -0.109413, z_c, rx, ry, rz], a, v)
    movel(p[x_c + 0.010440, y_c + -0.109441, z_c, rx, ry, rz], a, v)
    movel(p[x_c + 0.010533, y_c + -0.109473, z_c, rx, ry, rz], a, v)
    movel(p[x_c + 0.010626, y_c + -0.109507, z_c, rx, ry, rz], a, v)
    movel(p[x_c + 0.010720, y_c + -0.109544, z_c, rx, ry, rz], a, v)
    movel(p[x_c + 0.010815, y_c + -0.109585, z_c, rx, ry, rz], a, v)
    movel(p[x_c + 0.010910, y_c + -0.109629, z_c, rx, ry, rz], a, v)
    movel(p[x_c + 0.011007, y_c + -0.109676, z_c, rx, ry, rz], a, v)
    movel(p[x_c + 0.011103, y_c + -0.109726, z_c, rx, ry, rz], a, v)
    movel(p[x_c + 0.011201, y_c + -0.109780, z_c, rx, ry, rz], a, v)
    movel(p[x_c + 0.011299, y_c + -0.109837, z_c, rx, ry, rz], a, v)
    movel(p[x_c + 0.011399, y_c + -0.109897, z_c, rx, ry, rz], a, v)
    movel(p[x_c + 0.011499, y_c + -0.109961, z_c, rx, ry, rz], a, v)
    movel(p[x_c + 0.011600, y_c + -0.110028, z_c, rx, ry, rz], a, v)
    movel(p[x_c + 0.011703, y_c + -0.110098, z_c, rx, ry, rz], a, v)
    movel(p[x_c + 0.011806, y_c + -0.110172, z_c, rx, ry, rz], a, v)
    movel(p[x_c + 0.011911, y_c + -0.110250, z_c, rx, ry, rz], a, v)
    movel(p[x_c + 0.012017, y_c + -0.110331, z_c, rx, ry, rz], a, v)
    movel(p[x_c + 0.012124, y_c + -0.110416, z_c, rx, ry, rz], a, v)
    movel(p[x_c + 0.012233, y_c + -0.110504, z_c, rx, ry, rz], a, v)
    movel(p[x_c + 0.012342, y_c + -0.110596, z_c, rx, ry, rz], a, v)
    movel(p[x_c + 0.012454, y_c + -0.110692, z_c, rx, ry, rz], a, v)
    movel(p[x_c + 0.012567, y_c + -0.110791, z_c, rx, ry, rz], a, v)
    movel(p[x_c + 0.012681, y_c + -0.110894, z_c, rx, ry, rz], a, v)
    movel(p[x_c + 0.012797, y_c + -0.111001, z_c, rx, ry, rz], a, v)
    movel(p[x_c + 0.012915, y_c + -0.111112, z_c, rx, ry, rz], a, v)
    movel(p[x_c + 0.013034, y_c + -0.111226, z_c, rx, ry, rz], a, v)
    movel(p[x_c + 0.013156, y_c + -0.111345, z_c, rx, ry, rz], a, v)
    movel(p[x_c + 0.013279, y_c + -0.111467, z_c, rx, ry, rz], a, v)
    movel(p[x_c + 0.013403, y_c + -0.111593, z_c, rx, ry, rz], a, v)
    movel(p[x_c + 0.013530, y_c + -0.111723, z_c, rx, ry, rz], a, v)
    movel(p[x_c + 0.013659, y_c + -0.111857, z_c, rx, ry, rz], a, v)
    movel(p[x_c + 0.013790, y_c + -0.111996, z_c, rx, ry, rz], a, v)
    movel(p[x_c + 0.013923, y_c + -0.112138, z_c, rx, ry, rz], a, v)
    movel(p[x_c + 0.014058, y_c + -0.112284, z_c, rx, ry, rz], a, v)
    movel(p[x_c + 0.014058, y_c + -0.112284, z_c, rx, ry, rz], a, v)
    movel(p[x_c + 0.014235, y_c + -0.112475, z_c, rx, ry, rz], a, v)
    movel(p[x_c + 0.014409, y_c + -0.112661, z_c, rx, ry, rz], a, v)
    movel(p[x_c + 0.014581, y_c + -0.112841, z_c, rx, ry, rz], a, v)
    movel(p[x_c + 0.014751, y_c + -0.113015, z_c, rx, ry, rz], a, v)
    movel(p[x_c + 0.014919, y_c + -0.113184, z_c, rx, ry, rz], a, v)
    movel(p[x_c + 0.015085, y_c + -0.113348, z_c, rx, ry, rz], a, v)
    movel(p[x_c + 0.015248, y_c + -0.113506, z_c, rx, ry, rz], a, v)
    movel(p[x_c + 0.015410, y_c + -0.113658, z_c, rx, ry, rz], a, v)
    movel(p[x_c + 0.015570, y_c + -0.113806, z_c, rx, ry, rz], a, v)
    movel(p[x_c + 0.015728, y_c + -0.113948, z_c, rx, ry, rz], a, v)
    movel(p[x_c + 0.015885, y_c + -0.114084, z_c, rx, ry, rz], a, v)
    movel(p[x_c + 0.016039, y_c + -0.114216, z_c, rx, ry, rz], a, v)
    movel(p[x_c + 0.016192, y_c + -0.114342, z_c, rx, ry, rz], a, v)
    movel(p[x_c + 0.016344, y_c + -0.114463, z_c, rx, ry, rz], a, v)
    movel(p[x_c + 0.016494, y_c + -0.114579, z_c, rx, ry, rz], a, v)
    movel(p[x_c + 0.016643, y_c + -0.114689, z_c, rx, ry, rz], a, v)
    movel(p[x_c + 0.016791, y_c + -0.114795, z_c, rx, ry, rz], a, v)
    movel(p[x_c + 0.016937, y_c + -0.114896, z_c, rx, ry, rz], a, v)
    movel(p[x_c + 0.017083, y_c + -0.114991, z_c, rx, ry, rz], a, v)
    movel(p[x_c + 0.017227, y_c + -0.115082, z_c, rx, ry, rz], a, v)
    movel(p[x_c + 0.017370, y_c + -0.115167, z_c, rx, ry, rz], a, v)
    movel(p[x_c + 0.017512, y_c + -0.115248, z_c, rx, ry, rz], a, v)
    movel(p[x_c + 0.017654, y_c + -0.115324, z_c, rx, ry, rz], a, v)
    movel(p[x_c + 0.017795, y_c + -0.115395, z_c, rx, ry, rz], a, v)
    movel(p[x_c + 0.017935, y_c + -0.115461, z_c, rx, ry, rz], a, v)
    movel(p[x_c + 0.018074, y_c + -0.115523, z_c, rx, ry, rz], a, v)
    movel(p[x_c + 0.018213, y_c + -0.115579, z_c, rx, ry, rz], a, v)
    movel(p[x_c + 0.018352, y_c + -0.115631, z_c, rx, ry, rz], a, v)
    movel(p[x_c + 0.018490, y_c + -0.115679, z_c, rx, ry, rz], a, v)
    movel(p[x_c + 0.018628, y_c + -0.115721, z_c, rx, ry, rz], a, v)
    movel(p[x_c + 0.018765, y_c + -0.115760, z_c, rx, ry, rz], a, v)
    movel(p[x_c + 0.018902, y_c + -0.115793, z_c, rx, ry, rz], a, v)
    movel(p[x_c + 0.019040, y_c + -0.115822, z_c, rx, ry, rz], a, v)
    movel(p[x_c + 0.019177, y_c + -0.115847, z_c, rx, ry, rz], a, v)
    movel(p[x_c + 0.019314, y_c + -0.115867, z_c, rx, ry, rz], a, v)
    movel(p[x_c + 0.019452, y_c + -0.115882, z_c, rx, ry, rz], a, v)
    movel(p[x_c + 0.019589, y_c + -0.115894, z_c, rx, ry, rz], a, v)
    movel(p[x_c + 0.019727, y_c + -0.115901, z_c, rx, ry, rz], a, v)
    movel(p[x_c + 0.019865, y_c + -0.115903, z_c, rx, ry, rz], a, v)
    movel(p[x_c + 0.020004, y_c + -0.115901, z_c, rx, ry, rz], a, v)
    movel(p[x_c + 0.020143, y_c + -0.115896, z_c, rx, ry, rz], a, v)
    movel(p[x_c + 0.020283, y_c + -0.115885, z_c, rx, ry, rz], a, v)
    movel(p[x_c + 0.020423, y_c + -0.115871, z_c, rx, ry, rz], a, v)
    movel(p[x_c + 0.020564, y_c + -0.115853, z_c, rx, ry, rz], a, v)
    movel(p[x_c + 0.020706, y_c + -0.115830, z_c, rx, ry, rz], a, v)
    movel(p[x_c + 0.020849, y_c + -0.115803, z_c, rx, ry, rz], a, v)
    movel(p[x_c + 0.020993, y_c + -0.115773, z_c, rx, ry, rz], a, v)
    movel(p[x_c + 0.021137, y_c + -0.115738, z_c, rx, ry, rz], a, v)
    movel(p[x_c + 0.021283, y_c + -0.115699, z_c, rx, ry, rz], a, v)
    movel(p[x_c + 0.021283, y_c + -0.115699, z_c, rx, ry, rz], a, v)
    movel(p[x_c + 0.021283, y_c + -0.115699, z_c, rx, ry, rz], a, v)
    movel(p[x_c + 0.021283, y_c + -0.115699, z_c, rx, ry, rz], a, v)
    movel(p[x_c + 0.021283, y_c + -0.115699, z_c, rx, ry, rz], a, v)
    movel(p[x_c + 0.021283, y_c + -0.115699, z_c, rx, ry, rz], a, v)
    movel(p[x_c + 0.021283, y_c + -0.115699, z_c, rx, ry, rz], a, v)
    movel(p[x_c + 0.021283, y_c + -0.115699, z_c, rx, ry, rz], a, v)
    movel(p[x_c + 0.021283, y_c + -0.115699, z_c, rx, ry, rz], a, v)
    movel(p[x_c + 0.021283, y_c + -0.115699, z_c, rx, ry, rz], a, v)
    movel(p[x_c + 0.021283, y_c + -0.115699, z_c, rx, ry, rz], a, v)
    movel(p[x_c + 0.041364, y_c + -0.076176, z_c, rx, ry, rz], a, v)
    movel(p[x_c + 0.041364, y_c + -0.076176, z_c, rx, ry, rz], a, v)
    movel(p[x_c + 0.041364, y_c + -0.076176, z_c, rx, ry, rz], a, v)
    movel(p[x_c + 0.041364, y_c + -0.076176, z_c, rx, ry, rz], a, v)
    movel(p[x_c + 0.041364, y_c + -0.076176, z_c, rx, ry, rz], a, v)
    movel(p[x_c + 0.041364, y_c + -0.076176, z_c, rx, ry, rz], a, v)
    movel(p[x_c + 0.041364, y_c + -0.076176, z_c, rx, ry, rz], a, v)
    movel(p[x_c + 0.041364, y_c + -0.076176, z_c, rx, ry, rz], a, v)
    movel(p[x_c + 0.041364, y_c + -0.076176, z_c, rx, ry, rz], a, v)
    movel(p[x_c + 0.041364, y_c + -0.076176, z_c, rx, ry, rz], a, v)
    movel(p[x_c + 0.041364, y_c + -0.076176, z_c, rx, ry, rz], a, v)
    movel(p[x_c + 0.041394, y_c + -0.076114, z_c, rx, ry, rz], a, v)
    movel(p[x_c + 0.041422, y_c + -0.076047, z_c, rx, ry, rz], a, v)
    movel(p[x_c + 0.041448, y_c + -0.075975, z_c, rx, ry, rz], a, v)
    movel(p[x_c + 0.041471, y_c + -0.075897, z_c, rx, ry, rz], a, v)
    movel(p[x_c + 0.041492, y_c + -0.075813, z_c, rx, ry, rz], a, v)
    movel(p[x_c + 0.041511, y_c + -0.075725, z_c, rx, ry, rz], a, v)
    movel(p[x_c + 0.041528, y_c + -0.075630, z_c, rx, ry, rz], a, v)
    movel(p[x_c + 0.041542, y_c + -0.075531, z_c, rx, ry, rz], a, v)
    movel(p[x_c + 0.041554, y_c + -0.075426, z_c, rx, ry, rz], a, v)
    movel(p[x_c + 0.041564, y_c + -0.075317, z_c, rx, ry, rz], a, v)
    movel(p[x_c + 0.041571, y_c + -0.075202, z_c, rx, ry, rz], a, v)
    movel(p[x_c + 0.041576, y_c + -0.075081, z_c, rx, ry, rz], a, v)
    movel(p[x_c + 0.041579, y_c + -0.074956, z_c, rx, ry, rz], a, v)
    movel(p[x_c + 0.041580, y_c + -0.074826, z_c, rx, ry, rz], a, v)
    movel(p[x_c + 0.041578, y_c + -0.074691, z_c, rx, ry, rz], a, v)
    movel(p[x_c + 0.041574, y_c + -0.074550, z_c, rx, ry, rz], a, v)
    movel(p[x_c + 0.041568, y_c + -0.074405, z_c, rx, ry, rz], a, v)
    movel(p[x_c + 0.041560, y_c + -0.074255, z_c, rx, ry, rz], a, v)
    movel(p[x_c + 0.041549, y_c + -0.074100, z_c, rx, ry, rz], a, v)
    movel(p[x_c + 0.041537, y_c + -0.073940, z_c, rx, ry, rz], a, v)
    movel(p[x_c + 0.041522, y_c + -0.073775, z_c, rx, ry, rz], a, v)
    movel(p[x_c + 0.041504, y_c + -0.073606, z_c, rx, ry, rz], a, v)
    movel(p[x_c + 0.041485, y_c + -0.073432, z_c, rx, ry, rz], a, v)
    movel(p[x_c + 0.041463, y_c + -0.073253, z_c, rx, ry, rz], a, v)
    movel(p[x_c + 0.041440, y_c + -0.073069, z_c, rx, ry, rz], a, v)
    movel(p[x_c + 0.041414, y_c + -0.072881, z_c, rx, ry, rz], a, v)
    movel(p[x_c + 0.041385, y_c + -0.072689, z_c, rx, ry, rz], a, v)
    movel(p[x_c + 0.041355, y_c + -0.072491, z_c, rx, ry, rz], a, v)
    movel(p[x_c + 0.041323, y_c + -0.072290, z_c, rx, ry, rz], a, v)
    movel(p[x_c + 0.041288, y_c + -0.072084, z_c, rx, ry, rz], a, v)
    movel(p[x_c + 0.041251, y_c + -0.071873, z_c, rx, ry, rz], a, v)
    movel(p[x_c + 0.041212, y_c + -0.071658, z_c, rx, ry, rz], a, v)
    movel(p[x_c + 0.041171, y_c + -0.071439, z_c, rx, ry, rz], a, v)
    movel(p[x_c + 0.041127, y_c + -0.071215, z_c, rx, ry, rz], a, v)
    movel(p[x_c + 0.041082, y_c + -0.070987, z_c, rx, ry, rz], a, v)
    movel(p[x_c + 0.041034, y_c + -0.070755, z_c, rx, ry, rz], a, v)
    movel(p[x_c + 0.040984, y_c + -0.070519, z_c, rx, ry, rz], a, v)
    movel(p[x_c + 0.040932, y_c + -0.070278, z_c, rx, ry, rz], a, v)
    movel(p[x_c + 0.040878, y_c + -0.070034, z_c, rx, ry, rz], a, v)
    movel(p[x_c + 0.040822, y_c + -0.069785, z_c, rx, ry, rz], a, v)
    movel(p[x_c + 0.040764, y_c + -0.069533, z_c, rx, ry, rz], a, v)
    movel(p[x_c + 0.040703, y_c + -0.069276, z_c, rx, ry, rz], a, v)
    movel(p[x_c + 0.040641, y_c + -0.069015, z_c, rx, ry, rz], a, v)
    movel(p[x_c + 0.040576, y_c + -0.068751, z_c, rx, ry, rz], a, v)
    movel(p[x_c + 0.040509, y_c + -0.068482, z_c, rx, ry, rz], a, v)
    movel(p[x_c + 0.040440, y_c + -0.068210, z_c, rx, ry, rz], a, v)
    movel(p[x_c + 0.040369, y_c + -0.067934, z_c, rx, ry, rz], a, v)
    movel(p[x_c + 0.040296, y_c + -0.067654, z_c, rx, ry, rz], a, v)
    movel(p[x_c + 0.040221, y_c + -0.067370, z_c, rx, ry, rz], a, v)
    movel(p[x_c + 0.040221, y_c + -0.067370, z_c, rx, ry, rz], a, v)
    movel(p[x_c + 0.040019, y_c + -0.066610, z_c, rx, ry, rz], a, v)
    movel(p[x_c + 0.039823, y_c + -0.065865, z_c, rx, ry, rz], a, v)
    movel(p[x_c + 0.039632, y_c + -0.065135, z_c, rx, ry, rz], a, v)
    movel(p[x_c + 0.039447, y_c + -0.064418, z_c, rx, ry, rz], a, v)
    movel(p[x_c + 0.039267, y_c + -0.063715, z_c, rx, ry, rz], a, v)
    movel(p[x_c + 0.039092, y_c + -0.063025, z_c, rx, ry, rz], a, v)
    movel(p[x_c + 0.038923, y_c + -0.062347, z_c, rx, ry, rz], a, v)
    movel(p[x_c + 0.038758, y_c + -0.061681, z_c, rx, ry, rz], a, v)
    movel(p[x_c + 0.038599, y_c + -0.061026, z_c, rx, ry, rz], a, v)
    movel(p[x_c + 0.038444, y_c + -0.060382, z_c, rx, ry, rz], a, v)
    movel(p[x_c + 0.038295, y_c + -0.059748, z_c, rx, ry, rz], a, v)
    movel(p[x_c + 0.038150, y_c + -0.059125, z_c, rx, ry, rz], a, v)
    movel(p[x_c + 0.038009, y_c + -0.058510, z_c, rx, ry, rz], a, v)
    movel(p[x_c + 0.037874, y_c + -0.057904, z_c, rx, ry, rz], a, v)
    movel(p[x_c + 0.037742, y_c + -0.057306, z_c, rx, ry, rz], a, v)
    movel(p[x_c + 0.037615, y_c + -0.056716, z_c, rx, ry, rz], a, v)
    movel(p[x_c + 0.037493, y_c + -0.056133, z_c, rx, ry, rz], a, v)
    movel(p[x_c + 0.037374, y_c + -0.055557, z_c, rx, ry, rz], a, v)
    movel(p[x_c + 0.037260, y_c + -0.054987, z_c, rx, ry, rz], a, v)
    movel(p[x_c + 0.037150, y_c + -0.054422, z_c, rx, ry, rz], a, v)
    movel(p[x_c + 0.037043, y_c + -0.053863, z_c, rx, ry, rz], a, v)
    movel(p[x_c + 0.036941, y_c + -0.053308, z_c, rx, ry, rz], a, v)
    movel(p[x_c + 0.036842, y_c + -0.052757, z_c, rx, ry, rz], a, v)
    movel(p[x_c + 0.036747, y_c + -0.052210, z_c, rx, ry, rz], a, v)
    movel(p[x_c + 0.036655, y_c + -0.051665, z_c, rx, ry, rz], a, v)
    movel(p[x_c + 0.036568, y_c + -0.051124, z_c, rx, ry, rz], a, v)
    movel(p[x_c + 0.036483, y_c + -0.050584, z_c, rx, ry, rz], a, v)
    movel(p[x_c + 0.036402, y_c + -0.050045, z_c, rx, ry, rz], a, v)
    movel(p[x_c + 0.036324, y_c + -0.049508, z_c, rx, ry, rz], a, v)
    movel(p[x_c + 0.036249, y_c + -0.048971, z_c, rx, ry, rz], a, v)
    movel(p[x_c + 0.036177, y_c + -0.048433, z_c, rx, ry, rz], a, v)
    movel(p[x_c + 0.036109, y_c + -0.047895, z_c, rx, ry, rz], a, v)
    movel(p[x_c + 0.036043, y_c + -0.047356, z_c, rx, ry, rz], a, v)
    movel(p[x_c + 0.035980, y_c + -0.046816, z_c, rx, ry, rz], a, v)
    movel(p[x_c + 0.035920, y_c + -0.046273, z_c, rx, ry, rz], a, v)
    movel(p[x_c + 0.035862, y_c + -0.045727, z_c, rx, ry, rz], a, v)
    movel(p[x_c + 0.035807, y_c + -0.045178, z_c, rx, ry, rz], a, v)
    movel(p[x_c + 0.035754, y_c + -0.044626, z_c, rx, ry, rz], a, v)
    movel(p[x_c + 0.035704, y_c + -0.044069, z_c, rx, ry, rz], a, v)
    movel(p[x_c + 0.035656, y_c + -0.043507, z_c, rx, ry, rz], a, v)
    movel(p[x_c + 0.035610, y_c + -0.042940, z_c, rx, ry, rz], a, v)
    movel(p[x_c + 0.035567, y_c + -0.042368, z_c, rx, ry, rz], a, v)
    movel(p[x_c + 0.035525, y_c + -0.041788, z_c, rx, ry, rz], a, v)
    movel(p[x_c + 0.035485, y_c + -0.041202, z_c, rx, ry, rz], a, v)
    movel(p[x_c + 0.035447, y_c + -0.040609, z_c, rx, ry, rz], a, v)
    movel(p[x_c + 0.035411, y_c + -0.040008, z_c, rx, ry, rz], a, v)
    movel(p[x_c + 0.035377, y_c + -0.039398, z_c, rx, ry, rz], a, v)
    movel(p[x_c + 0.035344, y_c + -0.038779, z_c, rx, ry, rz], a, v)
    movel(p[x_c + 0.035313, y_c + -0.038151, z_c, rx, ry, rz], a, v)
    movel(p[x_c + 0.035313, y_c + -0.038151, z_c, rx, ry, rz], a, v)
    movel(p[x_c + 0.035293, y_c + -0.037707, z_c, rx, ry, rz], a, v)
    movel(p[x_c + 0.035275, y_c + -0.037250, z_c, rx, ry, rz], a, v)
    movel(p[x_c + 0.035260, y_c + -0.036778, z_c, rx, ry, rz], a, v)
    movel(p[x_c + 0.035248, y_c + -0.036293, z_c, rx, ry, rz], a, v)
    movel(p[x_c + 0.035237, y_c + -0.035795, z_c, rx, ry, rz], a, v)
    movel(p[x_c + 0.035229, y_c + -0.035285, z_c, rx, ry, rz], a, v)
    movel(p[x_c + 0.035224, y_c + -0.034764, z_c, rx, ry, rz], a, v)
    movel(p[x_c + 0.035220, y_c + -0.034232, z_c, rx, ry, rz], a, v)
    movel(p[x_c + 0.035219, y_c + -0.033689, z_c, rx, ry, rz], a, v)
    movel(p[x_c + 0.035220, y_c + -0.033137, z_c, rx, ry, rz], a, v)
    movel(p[x_c + 0.035223, y_c + -0.032575, z_c, rx, ry, rz], a, v)
    movel(p[x_c + 0.035229, y_c + -0.032005, z_c, rx, ry, rz], a, v)
    movel(p[x_c + 0.035236, y_c + -0.031426, z_c, rx, ry, rz], a, v)
    movel(p[x_c + 0.035246, y_c + -0.030841, z_c, rx, ry, rz], a, v)
    movel(p[x_c + 0.035257, y_c + -0.030248, z_c, rx, ry, rz], a, v)
    movel(p[x_c + 0.035271, y_c + -0.029648, z_c, rx, ry, rz], a, v)
    movel(p[x_c + 0.035286, y_c + -0.029043, z_c, rx, ry, rz], a, v)
    movel(p[x_c + 0.035304, y_c + -0.028433, z_c, rx, ry, rz], a, v)
    movel(p[x_c + 0.035324, y_c + -0.027818, z_c, rx, ry, rz], a, v)
    movel(p[x_c + 0.035345, y_c + -0.027199, z_c, rx, ry, rz], a, v)
    movel(p[x_c + 0.035369, y_c + -0.026576, z_c, rx, ry, rz], a, v)
    movel(p[x_c + 0.035394, y_c + -0.025950, z_c, rx, ry, rz], a, v)
    movel(p[x_c + 0.035421, y_c + -0.025322, z_c, rx, ry, rz], a, v)
    movel(p[x_c + 0.035450, y_c + -0.024692, z_c, rx, ry, rz], a, v)
    movel(p[x_c + 0.035481, y_c + -0.024061, z_c, rx, ry, rz], a, v)
    movel(p[x_c + 0.035513, y_c + -0.023429, z_c, rx, ry, rz], a, v)
    movel(p[x_c + 0.035548, y_c + -0.022797, z_c, rx, ry, rz], a, v)
    movel(p[x_c + 0.035584, y_c + -0.022166, z_c, rx, ry, rz], a, v)
    movel(p[x_c + 0.035621, y_c + -0.021535, z_c, rx, ry, rz], a, v)
    movel(p[x_c + 0.035660, y_c + -0.020906, z_c, rx, ry, rz], a, v)
    movel(p[x_c + 0.035701, y_c + -0.020280, z_c, rx, ry, rz], a, v)
    movel(p[x_c + 0.035744, y_c + -0.019656, z_c, rx, ry, rz], a, v)
    movel(p[x_c + 0.035788, y_c + -0.019035, z_c, rx, ry, rz], a, v)
    movel(p[x_c + 0.035833, y_c + -0.018418, z_c, rx, ry, rz], a, v)
    movel(p[x_c + 0.035881, y_c + -0.017805, z_c, rx, ry, rz], a, v)
    movel(p[x_c + 0.035929, y_c + -0.017198, z_c, rx, ry, rz], a, v)
    movel(p[x_c + 0.035979, y_c + -0.016596, z_c, rx, ry, rz], a, v)
    movel(p[x_c + 0.036031, y_c + -0.016000, z_c, rx, ry, rz], a, v)
    movel(p[x_c + 0.036084, y_c + -0.015411, z_c, rx, ry, rz], a, v)
    movel(p[x_c + 0.036138, y_c + -0.014830, z_c, rx, ry, rz], a, v)
    movel(p[x_c + 0.036193, y_c + -0.014256, z_c, rx, ry, rz], a, v)
    movel(p[x_c + 0.036250, y_c + -0.013690, z_c, rx, ry, rz], a, v)
    movel(p[x_c + 0.036309, y_c + -0.013134, z_c, rx, ry, rz], a, v)
    movel(p[x_c + 0.036368, y_c + -0.012587, z_c, rx, ry, rz], a, v)
    movel(p[x_c + 0.036429, y_c + -0.012050, z_c, rx, ry, rz], a, v)
    movel(p[x_c + 0.036491, y_c + -0.011524, z_c, rx, ry, rz], a, v)
    movel(p[x_c + 0.036554, y_c + -0.011010, z_c, rx, ry, rz], a, v)
    movel(p[x_c + 0.036618, y_c + -0.010507, z_c, rx, ry, rz], a, v)
    movel(p[x_c + 0.036683, y_c + -0.010016, z_c, rx, ry, rz], a, v)
    movel(p[x_c + 0.036683, y_c + -0.010016, z_c, rx, ry, rz], a, v)
    movel(p[x_c + 0.036707, y_c + -0.009837, z_c, rx, ry, rz], a, v)
    movel(p[x_c + 0.036729, y_c + -0.009646, z_c, rx, ry, rz], a, v)
    movel(p[x_c + 0.036751, y_c + -0.009444, z_c, rx, ry, rz], a, v)
    movel(p[x_c + 0.036773, y_c + -0.009231, z_c, rx, ry, rz], a, v)
    movel(p[x_c + 0.036793, y_c + -0.009009, z_c, rx, ry, rz], a, v)
    movel(p[x_c + 0.036813, y_c + -0.008776, z_c, rx, ry, rz], a, v)
    movel(p[x_c + 0.036833, y_c + -0.008535, z_c, rx, ry, rz], a, v)
    movel(p[x_c + 0.036851, y_c + -0.008285, z_c, rx, ry, rz], a, v)
    movel(p[x_c + 0.036869, y_c + -0.008027, z_c, rx, ry, rz], a, v)
    movel(p[x_c + 0.036887, y_c + -0.007761, z_c, rx, ry, rz], a, v)
    movel(p[x_c + 0.036903, y_c + -0.007489, z_c, rx, ry, rz], a, v)
    movel(p[x_c + 0.036919, y_c + -0.007211, z_c, rx, ry, rz], a, v)
    movel(p[x_c + 0.036934, y_c + -0.006926, z_c, rx, ry, rz], a, v)
    movel(p[x_c + 0.036949, y_c + -0.006636, z_c, rx, ry, rz], a, v)
    movel(p[x_c + 0.036962, y_c + -0.006342, z_c, rx, ry, rz], a, v)
    movel(p[x_c + 0.036975, y_c + -0.006043, z_c, rx, ry, rz], a, v)
    movel(p[x_c + 0.036987, y_c + -0.005741, z_c, rx, ry, rz], a, v)
    movel(p[x_c + 0.036999, y_c + -0.005436, z_c, rx, ry, rz], a, v)
    movel(p[x_c + 0.037009, y_c + -0.005128, z_c, rx, ry, rz], a, v)
    movel(p[x_c + 0.037019, y_c + -0.004818, z_c, rx, ry, rz], a, v)
    movel(p[x_c + 0.037028, y_c + -0.004507, z_c, rx, ry, rz], a, v)
    movel(p[x_c + 0.037036, y_c + -0.004194, z_c, rx, ry, rz], a, v)
    movel(p[x_c + 0.037043, y_c + -0.003882, z_c, rx, ry, rz], a, v)
    movel(p[x_c + 0.037050, y_c + -0.003569, z_c, rx, ry, rz], a, v)
    movel(p[x_c + 0.037055, y_c + -0.003257, z_c, rx, ry, rz], a, v)
    movel(p[x_c + 0.037060, y_c + -0.002946, z_c, rx, ry, rz], a, v)
    movel(p[x_c + 0.037064, y_c + -0.002637, z_c, rx, ry, rz], a, v)
    movel(p[x_c + 0.037067, y_c + -0.002331, z_c, rx, ry, rz], a, v)
    movel(p[x_c + 0.037069, y_c + -0.002027, z_c, rx, ry, rz], a, v)
    movel(p[x_c + 0.037070, y_c + -0.001727, z_c, rx, ry, rz], a, v)
    movel(p[x_c + 0.037070, y_c + -0.001430, z_c, rx, ry, rz], a, v)
    movel(p[x_c + 0.037070, y_c + -0.001138, z_c, rx, ry, rz], a, v)
    movel(p[x_c + 0.037068, y_c + -0.000851, z_c, rx, ry, rz], a, v)
    movel(p[x_c + 0.037066, y_c + -0.000569, z_c, rx, ry, rz], a, v)
    movel(p[x_c + 0.037062, y_c + -0.000294, z_c, rx, ry, rz], a, v)
    movel(p[x_c + 0.037058, y_c + -0.000025, z_c, rx, ry, rz], a, v)
    movel(p[x_c + 0.037053, y_c + 0.000236, z_c, rx, ry, rz], a, v)
    movel(p[x_c + 0.037046, y_c + 0.000490, z_c, rx, ry, rz], a, v)
    movel(p[x_c + 0.037039, y_c + 0.000736, z_c, rx, ry, rz], a, v)
    movel(p[x_c + 0.037031, y_c + 0.000973, z_c, rx, ry, rz], a, v)
    movel(p[x_c + 0.037021, y_c + 0.001201, z_c, rx, ry, rz], a, v)
    movel(p[x_c + 0.037011, y_c + 0.001418, z_c, rx, ry, rz], a, v)
    movel(p[x_c + 0.037000, y_c + 0.001626, z_c, rx, ry, rz], a, v)
    movel(p[x_c + 0.036987, y_c + 0.001822, z_c, rx, ry, rz], a, v)
    movel(p[x_c + 0.036974, y_c + 0.002007, z_c, rx, ry, rz], a, v)
    movel(p[x_c + 0.036960, y_c + 0.002180, z_c, rx, ry, rz], a, v)
    movel(p[x_c + 0.036944, y_c + 0.002340, z_c, rx, ry, rz], a, v)
    movel(p[x_c + 0.036927, y_c + 0.002487, z_c, rx, ry, rz], a, v)
    movel(p[x_c + 0.036910, y_c + 0.002621, z_c, rx, ry, rz], a, v)
    movel(p[x_c + 0.036910, y_c + 0.002621, z_c, rx, ry, rz], a, v)
    movel(p[x_c + 0.036887, y_c + 0.002775, z_c, rx, ry, rz], a, v)
    movel(p[x_c + 0.036863, y_c + 0.002929, z_c, rx, ry, rz], a, v)
    movel(p[x_c + 0.036837, y_c + 0.003084, z_c, rx, ry, rz], a, v)
    movel(p[x_c + 0.036810, y_c + 0.003239, z_c, rx, ry, rz], a, v)
    movel(p[x_c + 0.036782, y_c + 0.003395, z_c, rx, ry, rz], a, v)
    movel(p[x_c + 0.036752, y_c + 0.003551, z_c, rx, ry, rz], a, v)
    movel(p[x_c + 0.036721, y_c + 0.003708, z_c, rx, ry, rz], a, v)
    movel(p[x_c + 0.036688, y_c + 0.003866, z_c, rx, ry, rz], a, v)
    movel(p[x_c + 0.036654, y_c + 0.004024, z_c, rx, ry, rz], a, v)
    movel(p[x_c + 0.036618, y_c + 0.004183, z_c, rx, ry, rz], a, v)
    movel(p[x_c + 0.036581, y_c + 0.004342, z_c, rx, ry, rz], a, v)
    movel(p[x_c + 0.036543, y_c + 0.004502, z_c, rx, ry, rz], a, v)
    movel(p[x_c + 0.036503, y_c + 0.004662, z_c, rx, ry, rz], a, v)
    movel(p[x_c + 0.036462, y_c + 0.004823, z_c, rx, ry, rz], a, v)
    movel(p[x_c + 0.036419, y_c + 0.004985, z_c, rx, ry, rz], a, v)
    movel(p[x_c + 0.036374, y_c + 0.005147, z_c, rx, ry, rz], a, v)
    movel(p[x_c + 0.036329, y_c + 0.005310, z_c, rx, ry, rz], a, v)
    movel(p[x_c + 0.036282, y_c + 0.005474, z_c, rx, ry, rz], a, v)
    movel(p[x_c + 0.036233, y_c + 0.005638, z_c, rx, ry, rz], a, v)
    movel(p[x_c + 0.036183, y_c + 0.005803, z_c, rx, ry, rz], a, v)
    movel(p[x_c + 0.036131, y_c + 0.005969, z_c, rx, ry, rz], a, v)
    movel(p[x_c + 0.036078, y_c + 0.006135, z_c, rx, ry, rz], a, v)
    movel(p[x_c + 0.036024, y_c + 0.006302, z_c, rx, ry, rz], a, v)
    movel(p[x_c + 0.035968, y_c + 0.006470, z_c, rx, ry, rz], a, v)
    movel(p[x_c + 0.035911, y_c + 0.006638, z_c, rx, ry, rz], a, v)
    movel(p[x_c + 0.035852, y_c + 0.006807, z_c, rx, ry, rz], a, v)
    movel(p[x_c + 0.035791, y_c + 0.006977, z_c, rx, ry, rz], a, v)
    movel(p[x_c + 0.035729, y_c + 0.007148, z_c, rx, ry, rz], a, v)
    movel(p[x_c + 0.035666, y_c + 0.007319, z_c, rx, ry, rz], a, v)
    movel(p[x_c + 0.035601, y_c + 0.007491, z_c, rx, ry, rz], a, v)
    movel(p[x_c + 0.035535, y_c + 0.007664, z_c, rx, ry, rz], a, v)
    movel(p[x_c + 0.035467, y_c + 0.007838, z_c, rx, ry, rz], a, v)
    movel(p[x_c + 0.035398, y_c + 0.008012, z_c, rx, ry, rz], a, v)
    movel(p[x_c + 0.035327, y_c + 0.008187, z_c, rx, ry, rz], a, v)
    movel(p[x_c + 0.035254, y_c + 0.008363, z_c, rx, ry, rz], a, v)
    movel(p[x_c + 0.035181, y_c + 0.008540, z_c, rx, ry, rz], a, v)
    movel(p[x_c + 0.035105, y_c + 0.008717, z_c, rx, ry, rz], a, v)
    movel(p[x_c + 0.035028, y_c + 0.008896, z_c, rx, ry, rz], a, v)
    movel(p[x_c + 0.034950, y_c + 0.009075, z_c, rx, ry, rz], a, v)
    movel(p[x_c + 0.034870, y_c + 0.009255, z_c, rx, ry, rz], a, v)
    movel(p[x_c + 0.034788, y_c + 0.009436, z_c, rx, ry, rz], a, v)
    movel(p[x_c + 0.034705, y_c + 0.009618, z_c, rx, ry, rz], a, v)
    movel(p[x_c + 0.034621, y_c + 0.009801, z_c, rx, ry, rz], a, v)
    movel(p[x_c + 0.034535, y_c + 0.009984, z_c, rx, ry, rz], a, v)
    movel(p[x_c + 0.034447, y_c + 0.010169, z_c, rx, ry, rz], a, v)
    movel(p[x_c + 0.034358, y_c + 0.010354, z_c, rx, ry, rz], a, v)
    movel(p[x_c + 0.034267, y_c + 0.010540, z_c, rx, ry, rz], a, v)
    movel(p[x_c + 0.034175, y_c + 0.010727, z_c, rx, ry, rz], a, v)
    movel(p[x_c + 0.034081, y_c + 0.010915, z_c, rx, ry, rz], a, v)
    movel(p[x_c + 0.034081, y_c + 0.010915, z_c, rx, ry, rz], a, v)
    movel(p[x_c + 0.033909, y_c + 0.011259, z_c, rx, ry, rz], a, v)
    movel(p[x_c + 0.033739, y_c + 0.011602, z_c, rx, ry, rz], a, v)
    movel(p[x_c + 0.033570, y_c + 0.011943, z_c, rx, ry, rz], a, v)
    movel(p[x_c + 0.033402, y_c + 0.012284, z_c, rx, ry, rz], a, v)
    movel(p[x_c + 0.033236, y_c + 0.012623, z_c, rx, ry, rz], a, v)
    movel(p[x_c + 0.033072, y_c + 0.012962, z_c, rx, ry, rz], a, v)
    movel(p[x_c + 0.032908, y_c + 0.013299, z_c, rx, ry, rz], a, v)
    movel(p[x_c + 0.032746, y_c + 0.013636, z_c, rx, ry, rz], a, v)
    movel(p[x_c + 0.032586, y_c + 0.013973, z_c, rx, ry, rz], a, v)
    movel(p[x_c + 0.032426, y_c + 0.014309, z_c, rx, ry, rz], a, v)
    movel(p[x_c + 0.032268, y_c + 0.014644, z_c, rx, ry, rz], a, v)
    movel(p[x_c + 0.032111, y_c + 0.014979, z_c, rx, ry, rz], a, v)
    movel(p[x_c + 0.031955, y_c + 0.015314, z_c, rx, ry, rz], a, v)
    movel(p[x_c + 0.031801, y_c + 0.015649, z_c, rx, ry, rz], a, v)
    movel(p[x_c + 0.031647, y_c + 0.015984, z_c, rx, ry, rz], a, v)
    movel(p[x_c + 0.031494, y_c + 0.016319, z_c, rx, ry, rz], a, v)
    movel(p[x_c + 0.031342, y_c + 0.016654, z_c, rx, ry, rz], a, v)
    movel(p[x_c + 0.031191, y_c + 0.016989, z_c, rx, ry, rz], a, v)
    movel(p[x_c + 0.031041, y_c + 0.017325, z_c, rx, ry, rz], a, v)
    movel(p[x_c + 0.030892, y_c + 0.017661, z_c, rx, ry, rz], a, v)
    movel(p[x_c + 0.030743, y_c + 0.017998, z_c, rx, ry, rz], a, v)
    movel(p[x_c + 0.030596, y_c + 0.018335, z_c, rx, ry, rz], a, v)
    movel(p[x_c + 0.030449, y_c + 0.018673, z_c, rx, ry, rz], a, v)
    movel(p[x_c + 0.030302, y_c + 0.019012, z_c, rx, ry, rz], a, v)
    movel(p[x_c + 0.030157, y_c + 0.019353, z_c, rx, ry, rz], a, v)
    movel(p[x_c + 0.030011, y_c + 0.019694, z_c, rx, ry, rz], a, v)
    movel(p[x_c + 0.029867, y_c + 0.020036, z_c, rx, ry, rz], a, v)
    movel(p[x_c + 0.029723, y_c + 0.020380, z_c, rx, ry, rz], a, v)
    movel(p[x_c + 0.029579, y_c + 0.020725, z_c, rx, ry, rz], a, v)
    movel(p[x_c + 0.029435, y_c + 0.021071, z_c, rx, ry, rz], a, v)
    movel(p[x_c + 0.029292, y_c + 0.021419, z_c, rx, ry, rz], a, v)
    movel(p[x_c + 0.029150, y_c + 0.021769, z_c, rx, ry, rz], a, v)
    movel(p[x_c + 0.029007, y_c + 0.022120, z_c, rx, ry, rz], a, v)
    movel(p[x_c + 0.028865, y_c + 0.022473, z_c, rx, ry, rz], a, v)
    movel(p[x_c + 0.028723, y_c + 0.022829, z_c, rx, ry, rz], a, v)
    movel(p[x_c + 0.028582, y_c + 0.023186, z_c, rx, ry, rz], a, v)
    movel(p[x_c + 0.028440, y_c + 0.023545, z_c, rx, ry, rz], a, v)
    movel(p[x_c + 0.028298, y_c + 0.023907, z_c, rx, ry, rz], a, v)
    movel(p[x_c + 0.028157, y_c + 0.024271, z_c, rx, ry, rz], a, v)
    movel(p[x_c + 0.028015, y_c + 0.024638, z_c, rx, ry, rz], a, v)
    movel(p[x_c + 0.027873, y_c + 0.025007, z_c, rx, ry, rz], a, v)
    movel(p[x_c + 0.027731, y_c + 0.025378, z_c, rx, ry, rz], a, v)
    movel(p[x_c + 0.027589, y_c + 0.025753, z_c, rx, ry, rz], a, v)
    movel(p[x_c + 0.027447, y_c + 0.026130, z_c, rx, ry, rz], a, v)
    movel(p[x_c + 0.027305, y_c + 0.026510, z_c, rx, ry, rz], a, v)
    movel(p[x_c + 0.027162, y_c + 0.026894, z_c, rx, ry, rz], a, v)
    movel(p[x_c + 0.027019, y_c + 0.027280, z_c, rx, ry, rz], a, v)
    movel(p[x_c + 0.026876, y_c + 0.027670, z_c, rx, ry, rz], a, v)
    movel(p[x_c + 0.026732, y_c + 0.028063, z_c, rx, ry, rz], a, v)
    movel(p[x_c + 0.026732, y_c + 0.028063, z_c, rx, ry, rz], a, v)
    movel(p[x_c + 0.026640, y_c + 0.028316, z_c, rx, ry, rz], a, v)
    movel(p[x_c + 0.026549, y_c + 0.028562, z_c, rx, ry, rz], a, v)
    movel(p[x_c + 0.026461, y_c + 0.028801, z_c, rx, ry, rz], a, v)
    movel(p[x_c + 0.026375, y_c + 0.029034, z_c, rx, ry, rz], a, v)
    movel(p[x_c + 0.026291, y_c + 0.029261, z_c, rx, ry, rz], a, v)
    movel(p[x_c + 0.026208, y_c + 0.029481, z_c, rx, ry, rz], a, v)
    movel(p[x_c + 0.026128, y_c + 0.029696, z_c, rx, ry, rz], a, v)
    movel(p[x_c + 0.026049, y_c + 0.029905, z_c, rx, ry, rz], a, v)
    movel(p[x_c + 0.025971, y_c + 0.030108, z_c, rx, ry, rz], a, v)
    movel(p[x_c + 0.025896, y_c + 0.030305, z_c, rx, ry, rz], a, v)
    movel(p[x_c + 0.025821, y_c + 0.030497, z_c, rx, ry, rz], a, v)
    movel(p[x_c + 0.025749, y_c + 0.030684, z_c, rx, ry, rz], a, v)
    movel(p[x_c + 0.025677, y_c + 0.030866, z_c, rx, ry, rz], a, v)
    movel(p[x_c + 0.025607, y_c + 0.031044, z_c, rx, ry, rz], a, v)
    movel(p[x_c + 0.025538, y_c + 0.031216, z_c, rx, ry, rz], a, v)
    movel(p[x_c + 0.025470, y_c + 0.031384, z_c, rx, ry, rz], a, v)
    movel(p[x_c + 0.025403, y_c + 0.031548, z_c, rx, ry, rz], a, v)
    movel(p[x_c + 0.025337, y_c + 0.031707, z_c, rx, ry, rz], a, v)
    movel(p[x_c + 0.025272, y_c + 0.031863, z_c, rx, ry, rz], a, v)
    movel(p[x_c + 0.025208, y_c + 0.032014, z_c, rx, ry, rz], a, v)
    movel(p[x_c + 0.025144, y_c + 0.032162, z_c, rx, ry, rz], a, v)
    movel(p[x_c + 0.025082, y_c + 0.032306, z_c, rx, ry, rz], a, v)
    movel(p[x_c + 0.025019, y_c + 0.032447, z_c, rx, ry, rz], a, v)
    movel(p[x_c + 0.024958, y_c + 0.032584, z_c, rx, ry, rz], a, v)
    movel(p[x_c + 0.024897, y_c + 0.032719, z_c, rx, ry, rz], a, v)
    movel(p[x_c + 0.024836, y_c + 0.032851, z_c, rx, ry, rz], a, v)
    movel(p[x_c + 0.024775, y_c + 0.032980, z_c, rx, ry, rz], a, v)
    movel(p[x_c + 0.024715, y_c + 0.033106, z_c, rx, ry, rz], a, v)
    movel(p[x_c + 0.024655, y_c + 0.033230, z_c, rx, ry, rz], a, v)
    movel(p[x_c + 0.024595, y_c + 0.033351, z_c, rx, ry, rz], a, v)
    movel(p[x_c + 0.024535, y_c + 0.033471, z_c, rx, ry, rz], a, v)
    movel(p[x_c + 0.024475, y_c + 0.033589, z_c, rx, ry, rz], a, v)
    movel(p[x_c + 0.024414, y_c + 0.033705, z_c, rx, ry, rz], a, v)
    movel(p[x_c + 0.024354, y_c + 0.033819, z_c, rx, ry, rz], a, v)
    movel(p[x_c + 0.024293, y_c + 0.033932, z_c, rx, ry, rz], a, v)
    movel(p[x_c + 0.024232, y_c + 0.034043, z_c, rx, ry, rz], a, v)
    movel(p[x_c + 0.024171, y_c + 0.034154, z_c, rx, ry, rz], a, v)
    movel(p[x_c + 0.024109, y_c + 0.034263, z_c, rx, ry, rz], a, v)
    movel(p[x_c + 0.024046, y_c + 0.034372, z_c, rx, ry, rz], a, v)
    movel(p[x_c + 0.023983, y_c + 0.034480, z_c, rx, ry, rz], a, v)
    movel(p[x_c + 0.023919, y_c + 0.034588, z_c, rx, ry, rz], a, v)
    movel(p[x_c + 0.023854, y_c + 0.034695, z_c, rx, ry, rz], a, v)
    movel(p[x_c + 0.023788, y_c + 0.034802, z_c, rx, ry, rz], a, v)
    movel(p[x_c + 0.023722, y_c + 0.034909, z_c, rx, ry, rz], a, v)
    movel(p[x_c + 0.023654, y_c + 0.035017, z_c, rx, ry, rz], a, v)
    movel(p[x_c + 0.023585, y_c + 0.035124, z_c, rx, ry, rz], a, v)
    movel(p[x_c + 0.023516, y_c + 0.035232, z_c, rx, ry, rz], a, v)
    movel(p[x_c + 0.023444, y_c + 0.035341, z_c, rx, ry, rz], a, v)
    movel(p[x_c + 0.023372, y_c + 0.035451, z_c, rx, ry, rz], a, v)
    movel(p[x_c + 0.023372, y_c + 0.035451, z_c, rx, ry, rz], a, v)
    movel(p[x_c + 0.023274, y_c + 0.035596, z_c, rx, ry, rz], a, v)
    movel(p[x_c + 0.023176, y_c + 0.035737, z_c, rx, ry, rz], a, v)
    movel(p[x_c + 0.023078, y_c + 0.035874, z_c, rx, ry, rz], a, v)
    movel(p[x_c + 0.022980, y_c + 0.036007, z_c, rx, ry, rz], a, v)
    movel(p[x_c + 0.022881, y_c + 0.036137, z_c, rx, ry, rz], a, v)
    movel(p[x_c + 0.022781, y_c + 0.036262, z_c, rx, ry, rz], a, v)
    movel(p[x_c + 0.022682, y_c + 0.036384, z_c, rx, ry, rz], a, v)
    movel(p[x_c + 0.022582, y_c + 0.036502, z_c, rx, ry, rz], a, v)
    movel(p[x_c + 0.022482, y_c + 0.036616, z_c, rx, ry, rz], a, v)
    movel(p[x_c + 0.022381, y_c + 0.036726, z_c, rx, ry, rz], a, v)
    movel(p[x_c + 0.022280, y_c + 0.036833, z_c, rx, ry, rz], a, v)
    movel(p[x_c + 0.022178, y_c + 0.036935, z_c, rx, ry, rz], a, v)
    movel(p[x_c + 0.022076, y_c + 0.037034, z_c, rx, ry, rz], a, v)
    movel(p[x_c + 0.021974, y_c + 0.037129, z_c, rx, ry, rz], a, v)
    movel(p[x_c + 0.021871, y_c + 0.037220, z_c, rx, ry, rz], a, v)
    movel(p[x_c + 0.021768, y_c + 0.037308, z_c, rx, ry, rz], a, v)
    movel(p[x_c + 0.021664, y_c + 0.037392, z_c, rx, ry, rz], a, v)
    movel(p[x_c + 0.021559, y_c + 0.037471, z_c, rx, ry, rz], a, v)
    movel(p[x_c + 0.021454, y_c + 0.037548, z_c, rx, ry, rz], a, v)
    movel(p[x_c + 0.021349, y_c + 0.037620, z_c, rx, ry, rz], a, v)
    movel(p[x_c + 0.021243, y_c + 0.037689, z_c, rx, ry, rz], a, v)
    movel(p[x_c + 0.021136, y_c + 0.037754, z_c, rx, ry, rz], a, v)
    movel(p[x_c + 0.021029, y_c + 0.037815, z_c, rx, ry, rz], a, v)
    movel(p[x_c + 0.020921, y_c + 0.037872, z_c, rx, ry, rz], a, v)
    movel(p[x_c + 0.020813, y_c + 0.037926, z_c, rx, ry, rz], a, v)
    movel(p[x_c + 0.020704, y_c + 0.037976, z_c, rx, ry, rz], a, v)
    movel(p[x_c + 0.020594, y_c + 0.038023, z_c, rx, ry, rz], a, v)
    movel(p[x_c + 0.020483, y_c + 0.038065, z_c, rx, ry, rz], a, v)
    movel(p[x_c + 0.020372, y_c + 0.038104, z_c, rx, ry, rz], a, v)
    movel(p[x_c + 0.020260, y_c + 0.038140, z_c, rx, ry, rz], a, v)
    movel(p[x_c + 0.020148, y_c + 0.038172, z_c, rx, ry, rz], a, v)
    movel(p[x_c + 0.020034, y_c + 0.038200, z_c, rx, ry, rz], a, v)
    movel(p[x_c + 0.019920, y_c + 0.038224, z_c, rx, ry, rz], a, v)
    movel(p[x_c + 0.019805, y_c + 0.038245, z_c, rx, ry, rz], a, v)
    movel(p[x_c + 0.019690, y_c + 0.038262, z_c, rx, ry, rz], a, v)
    movel(p[x_c + 0.019573, y_c + 0.038275, z_c, rx, ry, rz], a, v)
    movel(p[x_c + 0.019456, y_c + 0.038285, z_c, rx, ry, rz], a, v)
    movel(p[x_c + 0.019338, y_c + 0.038292, z_c, rx, ry, rz], a, v)
    movel(p[x_c + 0.019219, y_c + 0.038294, z_c, rx, ry, rz], a, v)
    movel(p[x_c + 0.019099, y_c + 0.038293, z_c, rx, ry, rz], a, v)
    movel(p[x_c + 0.018979, y_c + 0.038289, z_c, rx, ry, rz], a, v)
    movel(p[x_c + 0.018857, y_c + 0.038281, z_c, rx, ry, rz], a, v)
    movel(p[x_c + 0.018735, y_c + 0.038269, z_c, rx, ry, rz], a, v)
    movel(p[x_c + 0.018611, y_c + 0.038254, z_c, rx, ry, rz], a, v)
    movel(p[x_c + 0.018487, y_c + 0.038235, z_c, rx, ry, rz], a, v)
    movel(p[x_c + 0.018362, y_c + 0.038213, z_c, rx, ry, rz], a, v)
    movel(p[x_c + 0.018235, y_c + 0.038187, z_c, rx, ry, rz], a, v)
    movel(p[x_c + 0.018108, y_c + 0.038157, z_c, rx, ry, rz], a, v)
    movel(p[x_c + 0.017980, y_c + 0.038125, z_c, rx, ry, rz], a, v)
    movel(p[x_c + 0.017980, y_c + 0.038125, z_c, rx, ry, rz], a, v)
    movel(p[x_c + 0.017894, y_c + 0.038101, z_c, rx, ry, rz], a, v)
    movel(p[x_c + 0.017809, y_c + 0.038076, z_c, rx, ry, rz], a, v)
    movel(p[x_c + 0.017726, y_c + 0.038049, z_c, rx, ry, rz], a, v)
    movel(p[x_c + 0.017644, y_c + 0.038022, z_c, rx, ry, rz], a, v)
    movel(p[x_c + 0.017563, y_c + 0.037994, z_c, rx, ry, rz], a, v)
    movel(p[x_c + 0.017484, y_c + 0.037964, z_c, rx, ry, rz], a, v)
    movel(p[x_c + 0.017406, y_c + 0.037934, z_c, rx, ry, rz], a, v)
    movel(p[x_c + 0.017330, y_c + 0.037902, z_c, rx, ry, rz], a, v)
    movel(p[x_c + 0.017255, y_c + 0.037870, z_c, rx, ry, rz], a, v)
    movel(p[x_c + 0.017182, y_c + 0.037836, z_c, rx, ry, rz], a, v)
    movel(p[x_c + 0.017111, y_c + 0.037802, z_c, rx, ry, rz], a, v)
    movel(p[x_c + 0.017040, y_c + 0.037767, z_c, rx, ry, rz], a, v)
    movel(p[x_c + 0.016972, y_c + 0.037730, z_c, rx, ry, rz], a, v)
    movel(p[x_c + 0.016905, y_c + 0.037693, z_c, rx, ry, rz], a, v)
    movel(p[x_c + 0.016840, y_c + 0.037655, z_c, rx, ry, rz], a, v)
    movel(p[x_c + 0.016776, y_c + 0.037615, z_c, rx, ry, rz], a, v)
    movel(p[x_c + 0.016714, y_c + 0.037575, z_c, rx, ry, rz], a, v)
    movel(p[x_c + 0.016653, y_c + 0.037534, z_c, rx, ry, rz], a, v)
    movel(p[x_c + 0.016594, y_c + 0.037493, z_c, rx, ry, rz], a, v)
    movel(p[x_c + 0.016537, y_c + 0.037450, z_c, rx, ry, rz], a, v)
    movel(p[x_c + 0.016482, y_c + 0.037407, z_c, rx, ry, rz], a, v)
    movel(p[x_c + 0.016428, y_c + 0.037363, z_c, rx, ry, rz], a, v)
    movel(p[x_c + 0.016376, y_c + 0.037318, z_c, rx, ry, rz], a, v)
    movel(p[x_c + 0.016325, y_c + 0.037272, z_c, rx, ry, rz], a, v)
    movel(p[x_c + 0.016277, y_c + 0.037225, z_c, rx, ry, rz], a, v)
    movel(p[x_c + 0.016230, y_c + 0.037178, z_c, rx, ry, rz], a, v)
    movel(p[x_c + 0.016185, y_c + 0.037130, z_c, rx, ry, rz], a, v)
    movel(p[x_c + 0.016142, y_c + 0.037082, z_c, rx, ry, rz], a, v)
    movel(p[x_c + 0.016101, y_c + 0.037032, z_c, rx, ry, rz], a, v)
    movel(p[x_c + 0.016061, y_c + 0.036982, z_c, rx, ry, rz], a, v)
    movel(p[x_c + 0.016024, y_c + 0.036931, z_c, rx, ry, rz], a, v)
    movel(p[x_c + 0.015988, y_c + 0.036880, z_c, rx, ry, rz], a, v)
    movel(p[x_c + 0.015954, y_c + 0.036828, z_c, rx, ry, rz], a, v)
    movel(p[x_c + 0.015922, y_c + 0.036776, z_c, rx, ry, rz], a, v)
    movel(p[x_c + 0.015892, y_c + 0.036723, z_c, rx, ry, rz], a, v)
    movel(p[x_c + 0.015864, y_c + 0.036669, z_c, rx, ry, rz], a, v)
    movel(p[x_c + 0.015838, y_c + 0.036615, z_c, rx, ry, rz], a, v)
    movel(p[x_c + 0.015814, y_c + 0.036560, z_c, rx, ry, rz], a, v)
    movel(p[x_c + 0.015792, y_c + 0.036505, z_c, rx, ry, rz], a, v)
    movel(p[x_c + 0.015772, y_c + 0.036449, z_c, rx, ry, rz], a, v)
    movel(p[x_c + 0.015754, y_c + 0.036392, z_c, rx, ry, rz], a, v)
    movel(p[x_c + 0.015738, y_c + 0.036336, z_c, rx, ry, rz], a, v)
    movel(p[x_c + 0.015724, y_c + 0.036278, z_c, rx, ry, rz], a, v)
    movel(p[x_c + 0.015712, y_c + 0.036221, z_c, rx, ry, rz], a, v)
    movel(p[x_c + 0.015703, y_c + 0.036163, z_c, rx, ry, rz], a, v)
    movel(p[x_c + 0.015695, y_c + 0.036104, z_c, rx, ry, rz], a, v)
    movel(p[x_c + 0.015690, y_c + 0.036045, z_c, rx, ry, rz], a, v)
    movel(p[x_c + 0.015687, y_c + 0.035986, z_c, rx, ry, rz], a, v)
    movel(p[x_c + 0.015685, y_c + 0.035926, z_c, rx, ry, rz], a, v)
    movel(p[x_c + 0.015685, y_c + 0.035926, z_c, rx, ry, rz], a, v)
    movel(p[x_c + 0.015686, y_c + 0.035852, z_c, rx, ry, rz], a, v)
    movel(p[x_c + 0.015689, y_c + 0.035779, z_c, rx, ry, rz], a, v)
    movel(p[x_c + 0.015693, y_c + 0.035705, z_c, rx, ry, rz], a, v)
    movel(p[x_c + 0.015700, y_c + 0.035631, z_c, rx, ry, rz], a, v)
    movel(p[x_c + 0.015708, y_c + 0.035556, z_c, rx, ry, rz], a, v)
    movel(p[x_c + 0.015718, y_c + 0.035482, z_c, rx, ry, rz], a, v)
    movel(p[x_c + 0.015730, y_c + 0.035407, z_c, rx, ry, rz], a, v)
    movel(p[x_c + 0.015744, y_c + 0.035332, z_c, rx, ry, rz], a, v)
    movel(p[x_c + 0.015759, y_c + 0.035256, z_c, rx, ry, rz], a, v)
    movel(p[x_c + 0.015777, y_c + 0.035180, z_c, rx, ry, rz], a, v)
    movel(p[x_c + 0.015798, y_c + 0.035103, z_c, rx, ry, rz], a, v)
    movel(p[x_c + 0.015820, y_c + 0.035026, z_c, rx, ry, rz], a, v)
    movel(p[x_c + 0.015844, y_c + 0.034947, z_c, rx, ry, rz], a, v)
    movel(p[x_c + 0.015871, y_c + 0.034868, z_c, rx, ry, rz], a, v)
    movel(p[x_c + 0.015900, y_c + 0.034789, z_c, rx, ry, rz], a, v)
    movel(p[x_c + 0.015931, y_c + 0.034708, z_c, rx, ry, rz], a, v)
    movel(p[x_c + 0.015964, y_c + 0.034626, z_c, rx, ry, rz], a, v)
    movel(p[x_c + 0.016000, y_c + 0.034543, z_c, rx, ry, rz], a, v)
    movel(p[x_c + 0.016038, y_c + 0.034460, z_c, rx, ry, rz], a, v)
    movel(p[x_c + 0.016079, y_c + 0.034375, z_c, rx, ry, rz], a, v)
    movel(p[x_c + 0.016122, y_c + 0.034288, z_c, rx, ry, rz], a, v)
    movel(p[x_c + 0.016167, y_c + 0.034201, z_c, rx, ry, rz], a, v)
    movel(p[x_c + 0.016215, y_c + 0.034112, z_c, rx, ry, rz], a, v)
    movel(p[x_c + 0.016266, y_c + 0.034022, z_c, rx, ry, rz], a, v)
    movel(p[x_c + 0.016319, y_c + 0.033930, z_c, rx, ry, rz], a, v)
    movel(p[x_c + 0.016375, y_c + 0.033836, z_c, rx, ry, rz], a, v)
    movel(p[x_c + 0.016434, y_c + 0.033741, z_c, rx, ry, rz], a, v)
    movel(p[x_c + 0.016495, y_c + 0.033645, z_c, rx, ry, rz], a, v)
    movel(p[x_c + 0.016560, y_c + 0.033546, z_c, rx, ry, rz], a, v)
    movel(p[x_c + 0.016627, y_c + 0.033446, z_c, rx, ry, rz], a, v)
    movel(p[x_c + 0.016696, y_c + 0.033344, z_c, rx, ry, rz], a, v)
    movel(p[x_c + 0.016769, y_c + 0.033240, z_c, rx, ry, rz], a, v)
    movel(p[x_c + 0.016845, y_c + 0.033134, z_c, rx, ry, rz], a, v)
    movel(p[x_c + 0.016923, y_c + 0.033025, z_c, rx, ry, rz], a, v)
    movel(p[x_c + 0.017005, y_c + 0.032915, z_c, rx, ry, rz], a, v)
    movel(p[x_c + 0.017090, y_c + 0.032802, z_c, rx, ry, rz], a, v)
    movel(p[x_c + 0.017177, y_c + 0.032688, z_c, rx, ry, rz], a, v)
    movel(p[x_c + 0.017268, y_c + 0.032570, z_c, rx, ry, rz], a, v)
    movel(p[x_c + 0.017362, y_c + 0.032451, z_c, rx, ry, rz], a, v)
    movel(p[x_c + 0.017459, y_c + 0.032329, z_c, rx, ry, rz], a, v)
    movel(p[x_c + 0.017560, y_c + 0.032204, z_c, rx, ry, rz], a, v)
    movel(p[x_c + 0.017663, y_c + 0.032077, z_c, rx, ry, rz], a, v)
    movel(p[x_c + 0.017770, y_c + 0.031947, z_c, rx, ry, rz], a, v)
    movel(p[x_c + 0.017880, y_c + 0.031814, z_c, rx, ry, rz], a, v)
    movel(p[x_c + 0.017994, y_c + 0.031679, z_c, rx, ry, rz], a, v)
    movel(p[x_c + 0.018111, y_c + 0.031541, z_c, rx, ry, rz], a, v)
    movel(p[x_c + 0.018232, y_c + 0.031400, z_c, rx, ry, rz], a, v)
    movel(p[x_c + 0.018356, y_c + 0.031255, z_c, rx, ry, rz], a, v)
    movel(p[x_c + 0.018483, y_c + 0.031108, z_c, rx, ry, rz], a, v)
    movel(p[x_c + 0.018483, y_c + 0.031108, z_c, rx, ry, rz], a, v)
    movel(p[x_c + 0.018639, y_c + 0.030929, z_c, rx, ry, rz], a, v)
    movel(p[x_c + 0.018790, y_c + 0.030754, z_c, rx, ry, rz], a, v)
    movel(p[x_c + 0.018938, y_c + 0.030583, z_c, rx, ry, rz], a, v)
    movel(p[x_c + 0.019081, y_c + 0.030416, z_c, rx, ry, rz], a, v)
    movel(p[x_c + 0.019221, y_c + 0.030252, z_c, rx, ry, rz], a, v)
    movel(p[x_c + 0.019357, y_c + 0.030093, z_c, rx, ry, rz], a, v)
    movel(p[x_c + 0.019490, y_c + 0.029937, z_c, rx, ry, rz], a, v)
    movel(p[x_c + 0.019619, y_c + 0.029785, z_c, rx, ry, rz], a, v)
    movel(p[x_c + 0.019744, y_c + 0.029635, z_c, rx, ry, rz], a, v)
    movel(p[x_c + 0.019866, y_c + 0.029489, z_c, rx, ry, rz], a, v)
    movel(p[x_c + 0.019985, y_c + 0.029346, z_c, rx, ry, rz], a, v)
    movel(p[x_c + 0.020101, y_c + 0.029207, z_c, rx, ry, rz], a, v)
    movel(p[x_c + 0.020213, y_c + 0.029069, z_c, rx, ry, rz], a, v)
    movel(p[x_c + 0.020323, y_c + 0.028935, z_c, rx, ry, rz], a, v)
    movel(p[x_c + 0.020430, y_c + 0.028803, z_c, rx, ry, rz], a, v)
    movel(p[x_c + 0.020534, y_c + 0.028674, z_c, rx, ry, rz], a, v)
    movel(p[x_c + 0.020635, y_c + 0.028546, z_c, rx, ry, rz], a, v)
    movel(p[x_c + 0.020734, y_c + 0.028422, z_c, rx, ry, rz], a, v)
    movel(p[x_c + 0.020830, y_c + 0.028299, z_c, rx, ry, rz], a, v)
    movel(p[x_c + 0.020924, y_c + 0.028178, z_c, rx, ry, rz], a, v)
    movel(p[x_c + 0.021016, y_c + 0.028058, z_c, rx, ry, rz], a, v)
    movel(p[x_c + 0.021105, y_c + 0.027941, z_c, rx, ry, rz], a, v)
    movel(p[x_c + 0.021192, y_c + 0.027825, z_c, rx, ry, rz], a, v)
    movel(p[x_c + 0.021277, y_c + 0.027711, z_c, rx, ry, rz], a, v)
    movel(p[x_c + 0.021360, y_c + 0.027597, z_c, rx, ry, rz], a, v)
    movel(p[x_c + 0.021442, y_c + 0.027485, z_c, rx, ry, rz], a, v)
    movel(p[x_c + 0.021521, y_c + 0.027374, z_c, rx, ry, rz], a, v)
    movel(p[x_c + 0.021599, y_c + 0.027264, z_c, rx, ry, rz], a, v)
    movel(p[x_c + 0.021675, y_c + 0.027155, z_c, rx, ry, rz], a, v)
    movel(p[x_c + 0.021750, y_c + 0.027046, z_c, rx, ry, rz], a, v)
    movel(p[x_c + 0.021824, y_c + 0.026938, z_c, rx, ry, rz], a, v)
    movel(p[x_c + 0.021896, y_c + 0.026830, z_c, rx, ry, rz], a, v)
    movel(p[x_c + 0.021967, y_c + 0.026723, z_c, rx, ry, rz], a, v)
    movel(p[x_c + 0.022037, y_c + 0.026615, z_c, rx, ry, rz], a, v)
    movel(p[x_c + 0.022105, y_c + 0.026508, z_c, rx, ry, rz], a, v)
    movel(p[x_c + 0.022173, y_c + 0.026401, z_c, rx, ry, rz], a, v)
    movel(p[x_c + 0.022240, y_c + 0.026293, z_c, rx, ry, rz], a, v)
    movel(p[x_c + 0.022307, y_c + 0.026185, z_c, rx, ry, rz], a, v)
    movel(p[x_c + 0.022373, y_c + 0.026077, z_c, rx, ry, rz], a, v)
    movel(p[x_c + 0.022438, y_c + 0.025967, z_c, rx, ry, rz], a, v)
    movel(p[x_c + 0.022502, y_c + 0.025858, z_c, rx, ry, rz], a, v)
    movel(p[x_c + 0.022567, y_c + 0.025747, z_c, rx, ry, rz], a, v)
    movel(p[x_c + 0.022631, y_c + 0.025635, z_c, rx, ry, rz], a, v)
    movel(p[x_c + 0.022695, y_c + 0.025523, z_c, rx, ry, rz], a, v)
    movel(p[x_c + 0.022759, y_c + 0.025408, z_c, rx, ry, rz], a, v)
    movel(p[x_c + 0.022822, y_c + 0.025293, z_c, rx, ry, rz], a, v)
    movel(p[x_c + 0.022886, y_c + 0.025176, z_c, rx, ry, rz], a, v)
    movel(p[x_c + 0.022951, y_c + 0.025058, z_c, rx, ry, rz], a, v)
    movel(p[x_c + 0.023015, y_c + 0.024937, z_c, rx, ry, rz], a, v)
    movel(p[x_c + 0.023015, y_c + 0.024937, z_c, rx, ry, rz], a, v)
    movel(p[x_c + 0.023226, y_c + 0.024533, z_c, rx, ry, rz], a, v)
    movel(p[x_c + 0.023429, y_c + 0.024125, z_c, rx, ry, rz], a, v)
    movel(p[x_c + 0.023626, y_c + 0.023713, z_c, rx, ry, rz], a, v)
    movel(p[x_c + 0.023815, y_c + 0.023296, z_c, rx, ry, rz], a, v)
    movel(p[x_c + 0.023997, y_c + 0.022873, z_c, rx, ry, rz], a, v)
    movel(p[x_c + 0.024172, y_c + 0.022444, z_c, rx, ry, rz], a, v)
    movel(p[x_c + 0.024340, y_c + 0.022009, z_c, rx, ry, rz], a, v)
    movel(p[x_c + 0.024501, y_c + 0.021568, z_c, rx, ry, rz], a, v)
    movel(p[x_c + 0.024655, y_c + 0.021119, z_c, rx, ry, rz], a, v)
    movel(p[x_c + 0.024802, y_c + 0.020662, z_c, rx, ry, rz], a, v)
    movel(p[x_c + 0.024942, y_c + 0.020198, z_c, rx, ry, rz], a, v)
    movel(p[x_c + 0.025075, y_c + 0.019725, z_c, rx, ry, rz], a, v)
    movel(p[x_c + 0.025201, y_c + 0.019243, z_c, rx, ry, rz], a, v)
    movel(p[x_c + 0.025321, y_c + 0.018751, z_c, rx, ry, rz], a, v)
    movel(p[x_c + 0.025434, y_c + 0.018249, z_c, rx, ry, rz], a, v)
    movel(p[x_c + 0.025540, y_c + 0.017737, z_c, rx, ry, rz], a, v)
    movel(p[x_c + 0.025639, y_c + 0.017215, z_c, rx, ry, rz], a, v)
    movel(p[x_c + 0.025732, y_c + 0.016680, z_c, rx, ry, rz], a, v)
    movel(p[x_c + 0.025818, y_c + 0.016135, z_c, rx, ry, rz], a, v)
    movel(p[x_c + 0.025898, y_c + 0.015576, z_c, rx, ry, rz], a, v)
    movel(p[x_c + 0.025970, y_c + 0.015006, z_c, rx, ry, rz], a, v)
    movel(p[x_c + 0.026037, y_c + 0.014422, z_c, rx, ry, rz], a, v)
    movel(p[x_c + 0.026097, y_c + 0.013824, z_c, rx, ry, rz], a, v)
    movel(p[x_c + 0.026150, y_c + 0.013213, z_c, rx, ry, rz], a, v)
    movel(p[x_c + 0.026197, y_c + 0.012587, z_c, rx, ry, rz], a, v)
    movel(p[x_c + 0.026238, y_c + 0.011946, z_c, rx, ry, rz], a, v)
    movel(p[x_c + 0.026272, y_c + 0.011290, z_c, rx, ry, rz], a, v)
    movel(p[x_c + 0.026300, y_c + 0.010617, z_c, rx, ry, rz], a, v)
    movel(p[x_c + 0.026321, y_c + 0.009929, z_c, rx, ry, rz], a, v)
    movel(p[x_c + 0.026337, y_c + 0.009224, z_c, rx, ry, rz], a, v)
    movel(p[x_c + 0.026346, y_c + 0.008501, z_c, rx, ry, rz], a, v)
    movel(p[x_c + 0.026349, y_c + 0.007761, z_c, rx, ry, rz], a, v)
    movel(p[x_c + 0.026346, y_c + 0.007003, z_c, rx, ry, rz], a, v)
    movel(p[x_c + 0.026336, y_c + 0.006226, z_c, rx, ry, rz], a, v)
    movel(p[x_c + 0.026321, y_c + 0.005430, z_c, rx, ry, rz], a, v)
    movel(p[x_c + 0.026299, y_c + 0.004614, z_c, rx, ry, rz], a, v)
    movel(p[x_c + 0.026272, y_c + 0.003779, z_c, rx, ry, rz], a, v)
    movel(p[x_c + 0.026238, y_c + 0.002923, z_c, rx, ry, rz], a, v)
    movel(p[x_c + 0.026199, y_c + 0.002046, z_c, rx, ry, rz], a, v)
    movel(p[x_c + 0.026154, y_c + 0.001148, z_c, rx, ry, rz], a, v)
    movel(p[x_c + 0.026102, y_c + 0.000229, z_c, rx, ry, rz], a, v)
    movel(p[x_c + 0.026045, y_c + -0.000713, z_c, rx, ry, rz], a, v)
    movel(p[x_c + 0.025982, y_c + -0.001678, z_c, rx, ry, rz], a, v)
    movel(p[x_c + 0.025914, y_c + -0.002666, z_c, rx, ry, rz], a, v)
    movel(p[x_c + 0.025839, y_c + -0.003677, z_c, rx, ry, rz], a, v)
    movel(p[x_c + 0.025759, y_c + -0.004713, z_c, rx, ry, rz], a, v)
    movel(p[x_c + 0.025673, y_c + -0.005773, z_c, rx, ry, rz], a, v)
    movel(p[x_c + 0.025582, y_c + -0.006858, z_c, rx, ry, rz], a, v)
    movel(p[x_c + 0.025485, y_c + -0.007968, z_c, rx, ry, rz], a, v)
    movel(p[x_c + 0.025485, y_c + -0.007968, z_c, rx, ry, rz], a, v)
    movel(p[x_c + 0.025379, y_c + -0.009199, z_c, rx, ry, rz], a, v)
    movel(p[x_c + 0.025282, y_c + -0.010419, z_c, rx, ry, rz], a, v)
    movel(p[x_c + 0.025194, y_c + -0.011628, z_c, rx, ry, rz], a, v)
    movel(p[x_c + 0.025115, y_c + -0.012827, z_c, rx, ry, rz], a, v)
    movel(p[x_c + 0.025044, y_c + -0.014015, z_c, rx, ry, rz], a, v)
    movel(p[x_c + 0.024983, y_c + -0.015193, z_c, rx, ry, rz], a, v)
    movel(p[x_c + 0.024930, y_c + -0.016361, z_c, rx, ry, rz], a, v)
    movel(p[x_c + 0.024886, y_c + -0.017520, z_c, rx, ry, rz], a, v)
    movel(p[x_c + 0.024851, y_c + -0.018670, z_c, rx, ry, rz], a, v)
    movel(p[x_c + 0.024825, y_c + -0.019811, z_c, rx, ry, rz], a, v)
    movel(p[x_c + 0.024808, y_c + -0.020944, z_c, rx, ry, rz], a, v)
    movel(p[x_c + 0.024800, y_c + -0.022068, z_c, rx, ry, rz], a, v)
    movel(p[x_c + 0.024802, y_c + -0.023184, z_c, rx, ry, rz], a, v)
    movel(p[x_c + 0.024812, y_c + -0.024292, z_c, rx, ry, rz], a, v)
    movel(p[x_c + 0.024831, y_c + -0.025393, z_c, rx, ry, rz], a, v)
    movel(p[x_c + 0.024860, y_c + -0.026486, z_c, rx, ry, rz], a, v)
    movel(p[x_c + 0.024897, y_c + -0.027573, z_c, rx, ry, rz], a, v)
    movel(p[x_c + 0.024944, y_c + -0.028652, z_c, rx, ry, rz], a, v)
    movel(p[x_c + 0.025000, y_c + -0.029726, z_c, rx, ry, rz], a, v)
    movel(p[x_c + 0.025066, y_c + -0.030793, z_c, rx, ry, rz], a, v)
    movel(p[x_c + 0.025141, y_c + -0.031855, z_c, rx, ry, rz], a, v)
    movel(p[x_c + 0.025225, y_c + -0.032911, z_c, rx, ry, rz], a, v)
    movel(p[x_c + 0.025318, y_c + -0.033962, z_c, rx, ry, rz], a, v)
    movel(p[x_c + 0.025421, y_c + -0.035007, z_c, rx, ry, rz], a, v)
    movel(p[x_c + 0.025533, y_c + -0.036048, z_c, rx, ry, rz], a, v)
    movel(p[x_c + 0.025655, y_c + -0.037085, z_c, rx, ry, rz], a, v)
    movel(p[x_c + 0.025786, y_c + -0.038117, z_c, rx, ry, rz], a, v)
    movel(p[x_c + 0.025926, y_c + -0.039146, z_c, rx, ry, rz], a, v)
    movel(p[x_c + 0.026076, y_c + -0.040171, z_c, rx, ry, rz], a, v)
    movel(p[x_c + 0.026236, y_c + -0.041192, z_c, rx, ry, rz], a, v)
    movel(p[x_c + 0.026406, y_c + -0.042211, z_c, rx, ry, rz], a, v)
    movel(p[x_c + 0.026585, y_c + -0.043227, z_c, rx, ry, rz], a, v)
    movel(p[x_c + 0.026773, y_c + -0.044240, z_c, rx, ry, rz], a, v)
    movel(p[x_c + 0.026972, y_c + -0.045251, z_c, rx, ry, rz], a, v)
    movel(p[x_c + 0.027180, y_c + -0.046260, z_c, rx, ry, rz], a, v)
    movel(p[x_c + 0.027397, y_c + -0.047267, z_c, rx, ry, rz], a, v)
    movel(p[x_c + 0.027625, y_c + -0.048273, z_c, rx, ry, rz], a, v)
    movel(p[x_c + 0.027862, y_c + -0.049278, z_c, rx, ry, rz], a, v)
    movel(p[x_c + 0.028109, y_c + -0.050282, z_c, rx, ry, rz], a, v)
    movel(p[x_c + 0.028367, y_c + -0.051286, z_c, rx, ry, rz], a, v)
    movel(p[x_c + 0.028634, y_c + -0.052289, z_c, rx, ry, rz], a, v)
    movel(p[x_c + 0.028910, y_c + -0.053292, z_c, rx, ry, rz], a, v)
    movel(p[x_c + 0.029197, y_c + -0.054296, z_c, rx, ry, rz], a, v)
    movel(p[x_c + 0.029494, y_c + -0.055300, z_c, rx, ry, rz], a, v)
    movel(p[x_c + 0.029801, y_c + -0.056305, z_c, rx, ry, rz], a, v)
    movel(p[x_c + 0.030118, y_c + -0.057311, z_c, rx, ry, rz], a, v)
    movel(p[x_c + 0.030445, y_c + -0.058318, z_c, rx, ry, rz], a, v)
    movel(p[x_c + 0.030782, y_c + -0.059327, z_c, rx, ry, rz], a, v)
    movel(p[x_c + 0.031129, y_c + -0.060338, z_c, rx, ry, rz], a, v)
    movel(p[x_c + 0.031129, y_c + -0.060338, z_c, rx, ry, rz], a, v)
    movel(p[x_c + 0.031356, y_c + -0.060982, z_c, rx, ry, rz], a, v)
    movel(p[x_c + 0.031587, y_c + -0.061619, z_c, rx, ry, rz], a, v)
    movel(p[x_c + 0.031820, y_c + -0.062248, z_c, rx, ry, rz], a, v)
    movel(p[x_c + 0.032057, y_c + -0.062870, z_c, rx, ry, rz], a, v)
    movel(p[x_c + 0.032296, y_c + -0.063483, z_c, rx, ry, rz], a, v)
    movel(p[x_c + 0.032537, y_c + -0.064088, z_c, rx, ry, rz], a, v)
    movel(p[x_c + 0.032780, y_c + -0.064684, z_c, rx, ry, rz], a, v)
    movel(p[x_c + 0.033025, y_c + -0.065270, z_c, rx, ry, rz], a, v)
    movel(p[x_c + 0.033272, y_c + -0.065847, z_c, rx, ry, rz], a, v)
    movel(p[x_c + 0.033520, y_c + -0.066413, z_c, rx, ry, rz], a, v)
    movel(p[x_c + 0.033768, y_c + -0.066969, z_c, rx, ry, rz], a, v)
    movel(p[x_c + 0.034018, y_c + -0.067513, z_c, rx, ry, rz], a, v)
    movel(p[x_c + 0.034268, y_c + -0.068047, z_c, rx, ry, rz], a, v)
    movel(p[x_c + 0.034518, y_c + -0.068568, z_c, rx, ry, rz], a, v)
    movel(p[x_c + 0.034768, y_c + -0.069077, z_c, rx, ry, rz], a, v)
    movel(p[x_c + 0.035018, y_c + -0.069573, z_c, rx, ry, rz], a, v)
    movel(p[x_c + 0.035267, y_c + -0.070056, z_c, rx, ry, rz], a, v)
    movel(p[x_c + 0.035516, y_c + -0.070526, z_c, rx, ry, rz], a, v)
    movel(p[x_c + 0.035763, y_c + -0.070982, z_c, rx, ry, rz], a, v)
    movel(p[x_c + 0.036009, y_c + -0.071423, z_c, rx, ry, rz], a, v)
    movel(p[x_c + 0.036253, y_c + -0.071850, z_c, rx, ry, rz], a, v)
    movel(p[x_c + 0.036495, y_c + -0.072262, z_c, rx, ry, rz], a, v)
    movel(p[x_c + 0.036736, y_c + -0.072658, z_c, rx, ry, rz], a, v)
    movel(p[x_c + 0.036974, y_c + -0.073038, z_c, rx, ry, rz], a, v)
    movel(p[x_c + 0.037209, y_c + -0.073402, z_c, rx, ry, rz], a, v)
    movel(p[x_c + 0.037441, y_c + -0.073749, z_c, rx, ry, rz], a, v)
    movel(p[x_c + 0.037670, y_c + -0.074079, z_c, rx, ry, rz], a, v)
    movel(p[x_c + 0.037895, y_c + -0.074391, z_c, rx, ry, rz], a, v)
    movel(p[x_c + 0.038117, y_c + -0.074686, z_c, rx, ry, rz], a, v)
    movel(p[x_c + 0.038335, y_c + -0.074962, z_c, rx, ry, rz], a, v)
    movel(p[x_c + 0.038548, y_c + -0.075219, z_c, rx, ry, rz], a, v)
    movel(p[x_c + 0.038757, y_c + -0.075457, z_c, rx, ry, rz], a, v)
    movel(p[x_c + 0.038961, y_c + -0.075675, z_c, rx, ry, rz], a, v)
    movel(p[x_c + 0.039161, y_c + -0.075874, z_c, rx, ry, rz], a, v)
    movel(p[x_c + 0.039354, y_c + -0.076052, z_c, rx, ry, rz], a, v)
    movel(p[x_c + 0.039543, y_c + -0.076209, z_c, rx, ry, rz], a, v)
    movel(p[x_c + 0.039725, y_c + -0.076345, z_c, rx, ry, rz], a, v)
    movel(p[x_c + 0.039902, y_c + -0.076460, z_c, rx, ry, rz], a, v)
    movel(p[x_c + 0.040071, y_c + -0.076552, z_c, rx, ry, rz], a, v)
    movel(p[x_c + 0.040235, y_c + -0.076622, z_c, rx, ry, rz], a, v)
    movel(p[x_c + 0.040391, y_c + -0.076670, z_c, rx, ry, rz], a, v)
    movel(p[x_c + 0.040541, y_c + -0.076693, z_c, rx, ry, rz], a, v)
    movel(p[x_c + 0.040683, y_c + -0.076694, z_c, rx, ry, rz], a, v)
    movel(p[x_c + 0.040817, y_c + -0.076670, z_c, rx, ry, rz], a, v)
    movel(p[x_c + 0.040943, y_c + -0.076622, z_c, rx, ry, rz], a, v)
    movel(p[x_c + 0.041061, y_c + -0.076549, z_c, rx, ry, rz], a, v)
    movel(p[x_c + 0.041171, y_c + -0.076450, z_c, rx, ry, rz], a, v)
    movel(p[x_c + 0.041272, y_c + -0.076326, z_c, rx, ry, rz], a, v)
    movel(p[x_c + 0.041364, y_c + -0.076176, z_c, rx, ry, rz], a, v)
    movel(p[x_c + 0.041364, y_c + -0.076176, z_c, rx, ry, rz], a, v)
    movel(p[x_c + 0.041364, y_c + -0.076176, z_c, rx, ry, rz], a, v)
    movel(p[x_c + 0.041364, y_c + -0.076176, z_c, rx, ry, rz], a, v)
    movel(p[x_c + 0.041364, y_c + -0.076176, z_c, rx, ry, rz], a, v)
    movel(p[x_c + 0.041364, y_c + -0.076176, z_c, rx, ry, rz], a, v)
    movel(p[x_c + 0.041364, y_c + -0.076176, z_c, rx, ry, rz], a, v)
    movel(p[x_c + 0.041364, y_c + -0.076176, z_c, rx, ry, rz], a, v)
    movel(p[x_c + 0.041364, y_c + -0.076176, z_c, rx, ry, rz], a, v)
    movel(p[x_c + 0.041364, y_c + -0.076176, z_c, rx, ry, rz], a, v)
    movel(p[x_c + 0.041364, y_c + -0.076176, z_c, rx, ry, rz], a, v)
    movel(p[x_c + 0.002172, y_c + 0.080094, z_c, rx, ry, rz], a, v)
    movel(p[x_c + 0.002172, y_c + 0.080094, z_c, rx, ry, rz], a, v)
    movel(p[x_c + 0.002172, y_c + 0.080094, z_c, rx, ry, rz], a, v)
    movel(p[x_c + 0.002172, y_c + 0.080094, z_c, rx, ry, rz], a, v)
    movel(p[x_c + 0.002172, y_c + 0.080094, z_c, rx, ry, rz], a, v)
    movel(p[x_c + 0.002172, y_c + 0.080094, z_c, rx, ry, rz], a, v)
    movel(p[x_c + 0.002172, y_c + 0.080094, z_c, rx, ry, rz], a, v)
    movel(p[x_c + 0.002172, y_c + 0.080094, z_c, rx, ry, rz], a, v)
    movel(p[x_c + 0.002172, y_c + 0.080094, z_c, rx, ry, rz], a, v)
    movel(p[x_c + 0.002172, y_c + 0.080094, z_c, rx, ry, rz], a, v)
    movel(p[x_c + 0.002172, y_c + 0.080094, z_c, rx, ry, rz], a, v)
    movel(p[x_c + 0.002347, y_c + 0.080127, z_c, rx, ry, rz], a, v)
    movel(p[x_c + 0.002520, y_c + 0.080164, z_c, rx, ry, rz], a, v)
    movel(p[x_c + 0.002692, y_c + 0.080204, z_c, rx, ry, rz], a, v)
    movel(p[x_c + 0.002863, y_c + 0.080246, z_c, rx, ry, rz], a, v)
    movel(p[x_c + 0.003032, y_c + 0.080291, z_c, rx, ry, rz], a, v)
    movel(p[x_c + 0.003200, y_c + 0.080340, z_c, rx, ry, rz], a, v)
    movel(p[x_c + 0.003367, y_c + 0.080390, z_c, rx, ry, rz], a, v)
    movel(p[x_c + 0.003532, y_c + 0.080444, z_c, rx, ry, rz], a, v)
    movel(p[x_c + 0.003696, y_c + 0.080500, z_c, rx, ry, rz], a, v)
    movel(p[x_c + 0.003858, y_c + 0.080559, z_c, rx, ry, rz], a, v)
    movel(p[x_c + 0.004019, y_c + 0.080621, z_c, rx, ry, rz], a, v)
    movel(p[x_c + 0.004178, y_c + 0.080685, z_c, rx, ry, rz], a, v)
    movel(p[x_c + 0.004335, y_c + 0.080752, z_c, rx, ry, rz], a, v)
    movel(p[x_c + 0.004491, y_c + 0.080822, z_c, rx, ry, rz], a, v)
    movel(p[x_c + 0.004645, y_c + 0.080894, z_c, rx, ry, rz], a, v)
    movel(p[x_c + 0.004797, y_c + 0.080969, z_c, rx, ry, rz], a, v)
    movel(p[x_c + 0.004948, y_c + 0.081046, z_c, rx, ry, rz], a, v)
    movel(p[x_c + 0.005097, y_c + 0.081126, z_c, rx, ry, rz], a, v)
    movel(p[x_c + 0.005244, y_c + 0.081208, z_c, rx, ry, rz], a, v)
    movel(p[x_c + 0.005389, y_c + 0.081293, z_c, rx, ry, rz], a, v)
    movel(p[x_c + 0.005532, y_c + 0.081380, z_c, rx, ry, rz], a, v)
    movel(p[x_c + 0.005673, y_c + 0.081469, z_c, rx, ry, rz], a, v)
    movel(p[x_c + 0.005812, y_c + 0.081561, z_c, rx, ry, rz], a, v)
    movel(p[x_c + 0.005950, y_c + 0.081655, z_c, rx, ry, rz], a, v)
    movel(p[x_c + 0.006085, y_c + 0.081751, z_c, rx, ry, rz], a, v)
    movel(p[x_c + 0.006218, y_c + 0.081850, z_c, rx, ry, rz], a, v)
    movel(p[x_c + 0.006349, y_c + 0.081951, z_c, rx, ry, rz], a, v)
    movel(p[x_c + 0.006477, y_c + 0.082054, z_c, rx, ry, rz], a, v)
    movel(p[x_c + 0.006604, y_c + 0.082160, z_c, rx, ry, rz], a, v)
    movel(p[x_c + 0.006728, y_c + 0.082267, z_c, rx, ry, rz], a, v)
    movel(p[x_c + 0.006850, y_c + 0.082377, z_c, rx, ry, rz], a, v)
    movel(p[x_c + 0.006970, y_c + 0.082489, z_c, rx, ry, rz], a, v)
    movel(p[x_c + 0.007088, y_c + 0.082603, z_c, rx, ry, rz], a, v)
    movel(p[x_c + 0.007203, y_c + 0.082719, z_c, rx, ry, rz], a, v)
    movel(p[x_c + 0.007315, y_c + 0.082837, z_c, rx, ry, rz], a, v)
    movel(p[x_c + 0.007425, y_c + 0.082957, z_c, rx, ry, rz], a, v)
    movel(p[x_c + 0.007533, y_c + 0.083079, z_c, rx, ry, rz], a, v)
    movel(p[x_c + 0.007638, y_c + 0.083204, z_c, rx, ry, rz], a, v)
    movel(p[x_c + 0.007741, y_c + 0.083330, z_c, rx, ry, rz], a, v)
    movel(p[x_c + 0.007841, y_c + 0.083458, z_c, rx, ry, rz], a, v)
    movel(p[x_c + 0.007938, y_c + 0.083588, z_c, rx, ry, rz], a, v)
    movel(p[x_c + 0.008033, y_c + 0.083719, z_c, rx, ry, rz], a, v)
    movel(p[x_c + 0.008124, y_c + 0.083853, z_c, rx, ry, rz], a, v)
    movel(p[x_c + 0.008214, y_c + 0.083988, z_c, rx, ry, rz], a, v)
    movel(p[x_c + 0.008300, y_c + 0.084126, z_c, rx, ry, rz], a, v)
    movel(p[x_c + 0.008384, y_c + 0.084265, z_c, rx, ry, rz], a, v)
    movel(p[x_c + 0.008464, y_c + 0.084405, z_c, rx, ry, rz], a, v)
    movel(p[x_c + 0.008542, y_c + 0.084548, z_c, rx, ry, rz], a, v)
    movel(p[x_c + 0.008617, y_c + 0.084692, z_c, rx, ry, rz], a, v)
    movel(p[x_c + 0.008617, y_c + 0.084692, z_c, rx, ry, rz], a, v)
    movel(p[x_c + 0.008658, y_c + 0.084775, z_c, rx, ry, rz], a, v)
    movel(p[x_c + 0.008699, y_c + 0.084862, z_c, rx, ry, rz], a, v)
    movel(p[x_c + 0.008740, y_c + 0.084952, z_c, rx, ry, rz], a, v)
    movel(p[x_c + 0.008781, y_c + 0.085045, z_c, rx, ry, rz], a, v)
    movel(p[x_c + 0.008821, y_c + 0.085140, z_c, rx, ry, rz], a, v)
    movel(p[x_c + 0.008860, y_c + 0.085239, z_c, rx, ry, rz], a, v)
    movel(p[x_c + 0.008900, y_c + 0.085341, z_c, rx, ry, rz], a, v)
    movel(p[x_c + 0.008939, y_c + 0.085445, z_c, rx, ry, rz], a, v)
    movel(p[x_c + 0.008977, y_c + 0.085551, z_c, rx, ry, rz], a, v)
    movel(p[x_c + 0.009016, y_c + 0.085660, z_c, rx, ry, rz], a, v)
    movel(p[x_c + 0.009053, y_c + 0.085772, z_c, rx, ry, rz], a, v)
    movel(p[x_c + 0.009090, y_c + 0.085885, z_c, rx, ry, rz], a, v)
    movel(p[x_c + 0.009127, y_c + 0.086000, z_c, rx, ry, rz], a, v)
    movel(p[x_c + 0.009163, y_c + 0.086118, z_c, rx, ry, rz], a, v)
    movel(p[x_c + 0.009199, y_c + 0.086237, z_c, rx, ry, rz], a, v)
    movel(p[x_c + 0.009234, y_c + 0.086358, z_c, rx, ry, rz], a, v)
    movel(p[x_c + 0.009268, y_c + 0.086480, z_c, rx, ry, rz], a, v)
    movel(p[x_c + 0.009302, y_c + 0.086604, z_c, rx, ry, rz], a, v)
    movel(p[x_c + 0.009335, y_c + 0.086729, z_c, rx, ry, rz], a, v)
    movel(p[x_c + 0.009367, y_c + 0.086855, z_c, rx, ry, rz], a, v)
    movel(p[x_c + 0.009398, y_c + 0.086982, z_c, rx, ry, rz], a, v)
    movel(p[x_c + 0.009429, y_c + 0.087111, z_c, rx, ry, rz], a, v)
    movel(p[x_c + 0.009459, y_c + 0.087240, z_c, rx, ry, rz], a, v)
    movel(p[x_c + 0.009488, y_c + 0.087370, z_c, rx, ry, rz], a, v)
    movel(p[x_c + 0.009517, y_c + 0.087500, z_c, rx, ry, rz], a, v)
    movel(p[x_c + 0.009544, y_c + 0.087631, z_c, rx, ry, rz], a, v)
    movel(p[x_c + 0.009571, y_c + 0.087762, z_c, rx, ry, rz], a, v)
    movel(p[x_c + 0.009597, y_c + 0.087894, z_c, rx, ry, rz], a, v)
    movel(p[x_c + 0.009621, y_c + 0.088026, z_c, rx, ry, rz], a, v)
    movel(p[x_c + 0.009645, y_c + 0.088157, z_c, rx, ry, rz], a, v)
    movel(p[x_c + 0.009668, y_c + 0.088289, z_c, rx, ry, rz], a, v)
    movel(p[x_c + 0.009690, y_c + 0.088420, z_c, rx, ry, rz], a, v)
    movel(p[x_c + 0.009710, y_c + 0.088551, z_c, rx, ry, rz], a, v)
    movel(p[x_c + 0.009730, y_c + 0.088682, z_c, rx, ry, rz], a, v)
    movel(p[x_c + 0.009749, y_c + 0.088812, z_c, rx, ry, rz], a, v)
    movel(p[x_c + 0.009766, y_c + 0.088941, z_c, rx, ry, rz], a, v)
    movel(p[x_c + 0.009783, y_c + 0.089069, z_c, rx, ry, rz], a, v)
    movel(p[x_c + 0.009798, y_c + 0.089197, z_c, rx, ry, rz], a, v)
    movel(p[x_c + 0.009812, y_c + 0.089323, z_c, rx, ry, rz], a, v)
    movel(p[x_c + 0.009825, y_c + 0.089448, z_c, rx, ry, rz], a, v)
    movel(p[x_c + 0.009836, y_c + 0.089572, z_c, rx, ry, rz], a, v)
    movel(p[x_c + 0.009846, y_c + 0.089695, z_c, rx, ry, rz], a, v)
    movel(p[x_c + 0.009855, y_c + 0.089816, z_c, rx, ry, rz], a, v)
    movel(p[x_c + 0.009863, y_c + 0.089935, z_c, rx, ry, rz], a, v)
    movel(p[x_c + 0.009869, y_c + 0.090053, z_c, rx, ry, rz], a, v)
    movel(p[x_c + 0.009874, y_c + 0.090168, z_c, rx, ry, rz], a, v)
    movel(p[x_c + 0.009878, y_c + 0.090282, z_c, rx, ry, rz], a, v)
    movel(p[x_c + 0.009880, y_c + 0.090394, z_c, rx, ry, rz], a, v)
    movel(p[x_c + 0.009880, y_c + 0.090503, z_c, rx, ry, rz], a, v)
    movel(p[x_c + 0.009880, y_c + 0.090503, z_c, rx, ry, rz], a, v)
    movel(p[x_c + 0.009878, y_c + 0.090710, z_c, rx, ry, rz], a, v)
    movel(p[x_c + 0.009872, y_c + 0.090923, z_c, rx, ry, rz], a, v)
    movel(p[x_c + 0.009863, y_c + 0.091141, z_c, rx, ry, rz], a, v)
    movel(p[x_c + 0.009851, y_c + 0.091365, z_c, rx, ry, rz], a, v)
    movel(p[x_c + 0.009835, y_c + 0.091592, z_c, rx, ry, rz], a, v)
    movel(p[x_c + 0.009816, y_c + 0.091825, z_c, rx, ry, rz], a, v)
    movel(p[x_c + 0.009794, y_c + 0.092062, z_c, rx, ry, rz], a, v)
    movel(p[x_c + 0.009769, y_c + 0.092303, z_c, rx, ry, rz], a, v)
    movel(p[x_c + 0.009741, y_c + 0.092547, z_c, rx, ry, rz], a, v)
    movel(p[x_c + 0.009709, y_c + 0.092796, z_c, rx, ry, rz], a, v)
    movel(p[x_c + 0.009675, y_c + 0.093048, z_c, rx, ry, rz], a, v)
    movel(p[x_c + 0.009638, y_c + 0.093303, z_c, rx, ry, rz], a, v)
    movel(p[x_c + 0.009598, y_c + 0.093560, z_c, rx, ry, rz], a, v)
    movel(p[x_c + 0.009555, y_c + 0.093821, z_c, rx, ry, rz], a, v)
    movel(p[x_c + 0.009509, y_c + 0.094084, z_c, rx, ry, rz], a, v)
    movel(p[x_c + 0.009461, y_c + 0.094350, z_c, rx, ry, rz], a, v)
    movel(p[x_c + 0.009410, y_c + 0.094617, z_c, rx, ry, rz], a, v)
    movel(p[x_c + 0.009357, y_c + 0.094886, z_c, rx, ry, rz], a, v)
    movel(p[x_c + 0.009301, y_c + 0.095157, z_c, rx, ry, rz], a, v)
    movel(p[x_c + 0.009242, y_c + 0.095429, z_c, rx, ry, rz], a, v)
    movel(p[x_c + 0.009182, y_c + 0.095703, z_c, rx, ry, rz], a, v)
    movel(p[x_c + 0.009119, y_c + 0.095977, z_c, rx, ry, rz], a, v)
    movel(p[x_c + 0.009053, y_c + 0.096251, z_c, rx, ry, rz], a, v)
    movel(p[x_c + 0.008986, y_c + 0.096527, z_c, rx, ry, rz], a, v)
    movel(p[x_c + 0.008916, y_c + 0.096802, z_c, rx, ry, rz], a, v)
    movel(p[x_c + 0.008844, y_c + 0.097078, z_c, rx, ry, rz], a, v)
    movel(p[x_c + 0.008770, y_c + 0.097353, z_c, rx, ry, rz], a, v)
    movel(p[x_c + 0.008695, y_c + 0.097627, z_c, rx, ry, rz], a, v)
    movel(p[x_c + 0.008617, y_c + 0.097901, z_c, rx, ry, rz], a, v)
    movel(p[x_c + 0.008537, y_c + 0.098174, z_c, rx, ry, rz], a, v)
    movel(p[x_c + 0.008456, y_c + 0.098446, z_c, rx, ry, rz], a, v)
    movel(p[x_c + 0.008373, y_c + 0.098716, z_c, rx, ry, rz], a, v)
    movel(p[x_c + 0.008288, y_c + 0.098985, z_c, rx, ry, rz], a, v)
    movel(p[x_c + 0.008201, y_c + 0.099252, z_c, rx, ry, rz], a, v)
    movel(p[x_c + 0.008113, y_c + 0.099517, z_c, rx, ry, rz], a, v)
    movel(p[x_c + 0.008024, y_c + 0.099779, z_c, rx, ry, rz], a, v)
    movel(p[x_c + 0.007933, y_c + 0.100039, z_c, rx, ry, rz], a, v)
    movel(p[x_c + 0.007840, y_c + 0.100296, z_c, rx, ry, rz], a, v)
    movel(p[x_c + 0.007747, y_c + 0.100550, z_c, rx, ry, rz], a, v)
    movel(p[x_c + 0.007651, y_c + 0.100801, z_c, rx, ry, rz], a, v)
    movel(p[x_c + 0.007555, y_c + 0.101049, z_c, rx, ry, rz], a, v)
    movel(p[x_c + 0.007458, y_c + 0.101292, z_c, rx, ry, rz], a, v)
    movel(p[x_c + 0.007359, y_c + 0.101532, z_c, rx, ry, rz], a, v)
    movel(p[x_c + 0.007259, y_c + 0.101768, z_c, rx, ry, rz], a, v)
    movel(p[x_c + 0.007159, y_c + 0.101999, z_c, rx, ry, rz], a, v)
    movel(p[x_c + 0.007057, y_c + 0.102225, z_c, rx, ry, rz], a, v)
    movel(p[x_c + 0.006955, y_c + 0.102447, z_c, rx, ry, rz], a, v)
    movel(p[x_c + 0.006851, y_c + 0.102664, z_c, rx, ry, rz], a, v)
    movel(p[x_c + 0.006747, y_c + 0.102875, z_c, rx, ry, rz], a, v)
    movel(p[x_c + 0.006747, y_c + 0.102875, z_c, rx, ry, rz], a, v)
    movel(p[x_c + 0.006570, y_c + 0.103225, z_c, rx, ry, rz], a, v)
    movel(p[x_c + 0.006391, y_c + 0.103572, z_c, rx, ry, rz], a, v)
    movel(p[x_c + 0.006210, y_c + 0.103914, z_c, rx, ry, rz], a, v)
    movel(p[x_c + 0.006026, y_c + 0.104253, z_c, rx, ry, rz], a, v)
    movel(p[x_c + 0.005841, y_c + 0.104589, z_c, rx, ry, rz], a, v)
    movel(p[x_c + 0.005654, y_c + 0.104920, z_c, rx, ry, rz], a, v)
    movel(p[x_c + 0.005465, y_c + 0.105248, z_c, rx, ry, rz], a, v)
    movel(p[x_c + 0.005274, y_c + 0.105571, z_c, rx, ry, rz], a, v)
    movel(p[x_c + 0.005082, y_c + 0.105891, z_c, rx, ry, rz], a, v)
    movel(p[x_c + 0.004888, y_c + 0.106206, z_c, rx, ry, rz], a, v)
    movel(p[x_c + 0.004692, y_c + 0.106518, z_c, rx, ry, rz], a, v)
    movel(p[x_c + 0.004494, y_c + 0.106825, z_c, rx, ry, rz], a, v)
    movel(p[x_c + 0.004295, y_c + 0.107128, z_c, rx, ry, rz], a, v)
    movel(p[x_c + 0.004095, y_c + 0.107427, z_c, rx, ry, rz], a, v)
    movel(p[x_c + 0.003893, y_c + 0.107721, z_c, rx, ry, rz], a, v)
    movel(p[x_c + 0.003689, y_c + 0.108011, z_c, rx, ry, rz], a, v)
    movel(p[x_c + 0.003484, y_c + 0.108296, z_c, rx, ry, rz], a, v)
    movel(p[x_c + 0.003278, y_c + 0.108577, z_c, rx, ry, rz], a, v)
